// POUs/Local/Objects/Primitive/FB_BACnet_INT
// Integer Value Object
{attribute 'enable_dynamic_creation'}
FUNCTION_BLOCK FB_BACnet_INT EXTENDS FB_BACnet_Object
VAR_INPUT CONSTANT PERSISTENT
	{region 'Operational Parameters'}
		{attribute 'parameterCategory':='Value'}
		nValue : DINT;
		{attribute 'parameterCategory':='Value'}
		eUnit : E_BA_Unit := E_BA_Unit.eOther_NoUnits;
	{endregion}
END_VAR
VAR_OUTPUT
	nPresVal : DINT;
END_VAR

IF bReady THEN
	nPresVal := nValue;
ELSE
	nPresVal := 0;
END_IF

SUPER^();

METHOD PROTECTED OnObjectStateChanged
SUPER^.OnObjectStateChanged();

CASE (tState) OF
	TCOM_STATE.TCOM_STATE_PREOP:
		// SyncHandler:
		RequestSyncHandlers(2, 2);

	TCOM_STATE.TCOM_STATE_SAFEOP:
		SyncProperty(E_BACnetPropIdentifier.PropPresentValue, SIZEOF(nValue), ADR(nValue), 0, eFullSync_InitPLC);
	
	TCOM_STATE.TCOM_STATE_OP:
		SyncProperty(E_BACnetPropIdentifier.PropUnits, SIZEOF(eUnit), ADR(eUnit), 0, eFullSync_InitPLC);
		
END_CASE
END_METHOD

METHOD FB_init : BOOL
VAR_INPUT
	bInitRetains : BOOL; // if TRUE, the retain variables are initialized (warm start / cold start)
	bInCopyCode : BOOL;  // if TRUE, the instance afterwards gets moved into the copy code (online change)
END_VAR
eObjectType := E_BACnetObjType.ObjIntegerValue;
END_METHOD

END_FUNCTION_BLOCK

// POUs/Local/Objects/Primitive/FB_BACnet_LAV
// Large AnalogValue Object
{attribute 'enable_dynamic_creation'}
FUNCTION_BLOCK FB_BACnet_LAV EXTENDS FB_BACnet_Object
VAR_INPUT CONSTANT PERSISTENT
	{region 'Operational Parameters'}
		{attribute 'parameterCategory':='Value'}
		fValue : LREAL;
		{attribute 'parameterCategory':='Value'}
		eUnit : E_BA_Unit := E_BA_Unit.eOther_NoUnits;
	{endregion}
END_VAR
VAR_OUTPUT
	fPresVal : LREAL;
END_VAR

IF bReady THEN
	fPresVal := fValue;
ELSE
	fPresVal := 0;
END_IF

SUPER^();

METHOD PROTECTED OnObjectStateChanged
SUPER^.OnObjectStateChanged();

CASE (tState) OF
	TCOM_STATE.TCOM_STATE_PREOP:
		// SyncHandler:
		RequestSyncHandlers(2, 2);

	TCOM_STATE.TCOM_STATE_SAFEOP:
		SyncProperty(E_BACnetPropIdentifier.PropPresentValue, SIZEOF(fValue), ADR(fValue), 0, eFullSync_InitPLC);
	
	TCOM_STATE.TCOM_STATE_OP:
		SyncProperty(E_BACnetPropIdentifier.PropUnits, SIZEOF(eUnit), ADR(eUnit), 0, eFullSync_InitPLC);
		
END_CASE
END_METHOD

METHOD FB_init : BOOL
VAR_INPUT
	bInitRetains : BOOL; // if TRUE, the retain variables are initialized (warm start / cold start)
	bInCopyCode : BOOL;  // if TRUE, the instance afterwards gets moved into the copy code (online change)
END_VAR
eObjectType := E_BACnetObjType.ObjLargeAnalogValue;
END_METHOD

END_FUNCTION_BLOCK

// POUs/Local/Objects/Primitive/FB_BACnet_String
// Integer Value Object
{attribute 'enable_dynamic_creation'}
FUNCTION_BLOCK FB_BACnet_String EXTENDS FB_BACnet_Object
VAR_INPUT CONSTANT PERSISTENT
	{region 'Operational Parameters'}
		{attribute 'parameterCategory':='Value'}
		{attribute 'TcEncoding':='UTF-8'}
		sValue : T_MaxString;
	{endregion}
END_VAR

SUPER^();

METHOD PROTECTED OnObjectStateChanged
SUPER^.OnObjectStateChanged();

CASE (tState) OF
	TCOM_STATE.TCOM_STATE_PREOP:
		// SyncHandler:
		RequestSyncHandlers(1, 1);

	TCOM_STATE.TCOM_STATE_SAFEOP:
		;
	
	TCOM_STATE.TCOM_STATE_OP:
		SyncProperty(E_BACnetPropIdentifier.PropDescription, SIZEOF(sValue), ADR(sValue), 0, eFullSync_InitPLC);
		
END_CASE
END_METHOD

METHOD FB_init : BOOL
VAR_INPUT
	bInitRetains : BOOL; // if TRUE, the retain variables are initialized (warm start / cold start)
	bInCopyCode : BOOL;  // if TRUE, the instance afterwards gets moved into the copy code (online change)
END_VAR
eObjectType := E_BACnetObjType.ObjCharacterStringValue;
END_METHOD

END_FUNCTION_BLOCK

// POUs/Local/Objects/Primitive/FB_BACnet_UINT
// Large AnalogValue Object
{attribute 'enable_dynamic_creation'}
FUNCTION_BLOCK FB_BACnet_UINT EXTENDS FB_BACnet_Object
VAR_INPUT CONSTANT PERSISTENT
	{region 'Operational Parameters'}
		{attribute 'parameterCategory':='Value'}
		nValue : DINT;
		{attribute 'parameterCategory':='Value'}
		eUnit : E_BA_Unit := E_BA_Unit.eOther_NoUnits;
	{endregion}
END_VAR
VAR_OUTPUT
	nPresVal : LREAL;
END_VAR

IF bReady THEN
	nPresVal := nValue;
ELSE
	nPresVal := 0;
END_IF

SUPER^();

METHOD PROTECTED OnObjectStateChanged
SUPER^.OnObjectStateChanged();

CASE (tState) OF
	TCOM_STATE.TCOM_STATE_PREOP:
		// SyncHandler:
		RequestSyncHandlers(2, 2);

	TCOM_STATE.TCOM_STATE_SAFEOP:
		SyncProperty(E_BACnetPropIdentifier.PropPresentValue, SIZEOF(nValue), ADR(nValue), 0, eFullSync_InitPLC);
	
	TCOM_STATE.TCOM_STATE_OP:
		SyncProperty(E_BACnetPropIdentifier.PropUnits, SIZEOF(eUnit), ADR(eUnit), 0, eFullSync_InitPLC);
		
END_CASE
END_METHOD

METHOD FB_init : BOOL
VAR_INPUT
	bInitRetains : BOOL; // if TRUE, the retain variables are initialized (warm start / cold start)
	bInCopyCode : BOOL;  // if TRUE, the instance afterwards gets moved into the copy code (online change)
END_VAR
eObjectType := E_BACnetObjType.ObjPositiveIntegerValue;
END_METHOD

END_FUNCTION_BLOCK

// POUs/Local/Objects/FB_BACnet_Acc_IO
// Accumulator Object
// - Terminal communication
{attribute 'pin_presentation_order_outputs' := 'nRawValue'}
FUNCTION_BLOCK FB_BACnet_Acc_IO EXTENDS FB_BACnet_BaseAcc
VAR_OUTPUT
	nPulseRate : UDINT;
END_VAR
VAR_INPUT CONSTANT PERSISTENT
	{region 'Variable Parameters'}
		{attribute 'parameterCategory':='Scale'}		  
		stScale : ST_BACnet_Scale;
		{attribute 'parameterCategory':='Scale'}		  	 
		stPrescale :  ST_BACnet_Prescale;
			  
		{attribute 'parameterCategory':='Value'}
		nValueSet : UDINT;
		{attribute 'parameterCategory':='Value'}
		{attribute 'parameterUnit':= 's'}	 
		nLimitMonitoringInterval : UDINT;		
	{endregion}
END_VAR
VAR PERSISTENT
	{region 'Output-Properties'}	
		{attribute 'parameterCategory':='Value'}
		nValueBeforeChange : UDINT;
		{attribute 'parameterCategory':='Value'}
		stValueChangeTime : ST_BA_DateTime;
	{endregion}
END_VAR
VAR
	{region 'Raw I/O'}
		nRawValue			AT %I*	: UINT;				// Bus terminal value
	{endregion}
END_VAR

SUPER^();

METHOD PROTECTED OnObjectStateChanged
CASE (tState) OF
	TCOM_STATE.TCOM_STATE_PREOP:
		// SyncHandler:
		RequestSyncHandlers(7, 5);
		
		WritePropertyUDInt(E_BACnetPropIdentifier.PropLimitMonitoringInverval, nLimitMonitoringInterval);
		
	TCOM_STATE.TCOM_STATE_SAFEOP:
		SyncProperty(E_BACnetPropIdentifier.PropRawIoAccumulatorUnsignedValue, SIZEOF(nRawValue), ADR(nRawValue), 0, eSync_ToSupplement);
		SyncProperty(E_BACnetPropIdentifier.PropPulseRate, SIZEOF(nPulseRate), ADR(nPulseRate), 0, eSync_FromSupplement);
		
	TCOM_STATE.TCOM_STATE_OP:
		SyncProperty(E_BACnetPropIdentifier.PropValueBeforeChange, SIZEOF(nValueBeforeChange), ADR(nValueBeforeChange), 0, eSync_FromSupplementInitPLC);
		SyncProperty(E_BACnetPropIdentifier.PropValueChangeTime, SIZEOF(stValueChangeTime), ADR(stValueChangeTime), 0, eSync_FromSupplementInitPLC);
		
		SyncProperty(E_BACnetPropIdentifier.PropLimitMonitoringInverval, SIZEOF(nLimitMonitoringInterval), ADR(nLimitMonitoringInterval), 0, eFullSync_InitPLC);
		SyncProperty(E_BACnetPropIdentifier.PropScale, SIZEOF(stScale), ADR(stScale), 0, eFullSync_InitPLC);
		SyncProperty(E_BACnetPropIdentifier.PropValueSet, SIZEOF(nValueSet), ADR(nValueSet), 0, eFullSync_InitPLC);		
		SyncProperty(E_BACnetPropIdentifier.PropPrescale, SIZEOF(stPrescale), ADR(stPrescale), 0, eFullSync_InitPLC);
		
END_CASE

SUPER^.OnObjectStateChanged();
END_METHOD

PROPERTY ValueBeforeChange : UDINT
GET
ValueBeforeChange := nValueBeforeChange;
END_GET
END_PROPERTY

PROPERTY ValueChangeTime : ST_BA_DateTime
GET
ValueChangeTime := stValueChangeTime;
END_GET
END_PROPERTY

END_FUNCTION_BLOCK

// POUs/Local/Objects/FB_BACnet_Acc_Raw
// Accumulator Object
// - Raw communication
{attribute 'pin_presentation_order_outputs' := 'fPresVal,bEvent,eRlbty'}
{attribute 'enable_dynamic_creation'}
FUNCTION_BLOCK FB_BACnet_Acc_Raw EXTENDS FB_BACnet_BaseAcc
VAR_INPUT
	{region 'Raw I/O'}
		nRawVal						: UINT;				// Raw value
	{endregion}
END_VAR
VAR_OUTPUT
	nPulseRate						: UDINT;
END_VAR
VAR_INPUT CONSTANT PERSISTENT
	{region 'Variable Parameters'}
		{attribute 'parameterCategory':='Scale'}		  
		stScale : ST_BACnet_Scale;
		{attribute 'parameterCategory':='Scale'}		  	 
		stPrescale :  ST_BACnet_Prescale;	
			  
		{attribute 'parameterCategory':='Value'}
		nValueSet : UDINT;
		{attribute 'parameterCategory':='Value'}
		{attribute 'parameterUnit':= 's'}	 
		nLimitMonitoringInterval : UDINT;		
	{endregion}
END_VAR
VAR PERSISTENT
	{region 'Output-Properties'}	
		nValueBeforeChange			: UDINT;
		stValueChangeTime			: ST_BA_DateTime;
	{endregion}
END_VAR

SUPER^();

METHOD PROTECTED OnObjectStateChanged
CASE (tState) OF
	TCOM_STATE.TCOM_STATE_PREOP:
		// SyncHandler:
		RequestSyncHandlers(8, 5);
		
		WritePropertyUDInt(E_BACnetPropIdentifier.PropLimitMonitoringInverval, nLimitMonitoringInterval);

	TCOM_STATE.TCOM_STATE_SAFEOP:
		SyncProperty(E_BACnetPropIdentifier.PropRawIoAccumulatorUnsignedValue, SIZEOF(nRawVal), ADR(nRawVal), 0, eSync_ToSupplement);
		SyncProperty(E_BACnetPropIdentifier.PropPulseRate, SIZEOF(nPulseRate), ADR(nPulseRate), 0, eSync_FromSupplement);
		
	TCOM_STATE.TCOM_STATE_OP:
		SyncProperty(E_BACnetPropIdentifier.PropValueBeforeChange, SIZEOF(nValueBeforeChange), ADR(nValueBeforeChange), 0, eSync_FromSupplementInitPLC);
		SyncProperty(E_BACnetPropIdentifier.PropValueChangeTime, SIZEOF(stValueChangeTime), ADR(stValueChangeTime), 0, eSync_FromSupplementInitPLC);
	
		SyncProperty(E_BACnetPropIdentifier.PropLimitMonitoringInverval, SIZEOF(nLimitMonitoringInterval), ADR(nLimitMonitoringInterval), 0, eFullSync_InitPLC);
		SyncProperty(E_BACnetPropIdentifier.PropScale, SIZEOF(stScale), ADR(stScale), 0, eFullSync_InitPLC);
		SyncProperty(E_BACnetPropIdentifier.PropValueSet, SIZEOF(nValueSet), ADR(nValueSet), 0, eFullSync_InitPLC);		
		SyncProperty(E_BACnetPropIdentifier.PropPrescale, SIZEOF(stPrescale), ADR(stPrescale), 0, eFullSync_InitPLC);
		
END_CASE

SUPER^.OnObjectStateChanged();
END_METHOD

END_FUNCTION_BLOCK

// POUs/Local/Objects/FB_BACnet_AI
// Analog Input Object
// - process value
{attribute 'pin_presentation_order_outputs' := 'fPresVal,bEvent,eRlbty'}
{attribute 'enable_dynamic_creation'}
FUNCTION_BLOCK FB_BACnet_AI EXTENDS FB_BACnet_BaseAI
VAR_INPUT
	fVal						: REAL;				// Process value
	eRlbtyPgm 					: E_BA_Reliability;
END_VAR

SUPER^();

METHOD PROTECTED OnObjectStateChanged
CASE (tState) OF
	TCOM_STATE.TCOM_STATE_PREOP:
		// SyncHandler:
		RequestSyncHandlers(0, 2);
		
		// Properties:
		EnableProperty(E_BACnetPropIdentifier.PropResolution, FALSE);
		EnableProperty(E_BACnetPropIdentifier.PropScaleOffset, FALSE);
	
	TCOM_STATE.TCOM_STATE_SAFEOP:
		SyncProperty(E_BACnetPropIdentifier.PropPresentValue, SIZEOF(fVal), ADR(fVal), 0, eSync_ToSupplement); 
		SyncProperty(E_BACnetPropIdentifier.PropReliability, SIZEOF(eRlbtyPgm), ADR(eRlbtyPgm), 0, eSync_ToSupplement);
		
	TCOM_STATE.TCOM_STATE_OP:
		;

END_CASE

SUPER^.OnObjectStateChanged();
END_METHOD

END_FUNCTION_BLOCK

// POUs/Local/Objects/FB_BACnet_AI_IO
// Analog Input Object
// - Terminal communication
{attribute 'pin_presentation_order_outputs' := 'fPresVal,bEvent,eRlbty'}
FUNCTION_BLOCK FB_BACnet_AI_IO EXTENDS FB_BACnet_BaseAI
VAR_INPUT CONSTANT PERSISTENT
	{region 'Fixed Parameters'}
		{attribute 'parameterCategory':='Hardware'}
		nIoBusNr : BYTE := 16#FF;
	{endregion}
	{region 'Variable Parameters'}
		{attribute 'parameterCategory':='Hardware'}
		fResolution : REAL := 0.1;
		{attribute 'parameterCategory':='Hardware'}
		fScaleOffset : REAL := 0;
	{endregion}
END_VAR
VAR
	{region 'Raw I/O'}
		nRawState			AT %I*	: USINT;			// Bus terminal state
		nRawValue			AT %I*	: INT;				// Bus terminal value
	{endregion}
END_VAR

SUPER^();

METHOD PROTECTED OnObjectStateChanged
CASE (tState) OF
	TCOM_STATE.TCOM_STATE_PREOP:
		// SyncHandler:
		RequestSyncHandlers(3, 4);

		IF (nIoBusNr <> 16#FF) THEN
			WritePropertyByte(E_BACnetPropIdentifier.PropIoBusNr, nIoBusNr);
		END_IF
		
	TCOM_STATE.TCOM_STATE_SAFEOP:
		SyncProperty(E_BACnetPropIdentifier.PropRawIoStateUSINT, SIZEOF(nRawState), ADR(nRawState), 0, eSync_ToSupplement);
		SyncProperty(E_BACnetPropIdentifier.PropRawIoAnalogValueINT, SIZEOF(nRawValue), ADR(nRawValue), 0, eSync_ToSupplement);
		
	TCOM_STATE.TCOM_STATE_OP:
		SyncProperty(E_BACnetPropIdentifier.PropResolution, SIZEOF(fResolution), ADR(fResolution), 0, eFullSync_InitPLC);
		SyncProperty(E_BACnetPropIdentifier.PropScaleOffset, SIZEOF(fScaleOffset), ADR(fScaleOffset), 0, eFullSync_InitPLC);
		
END_CASE

SUPER^.OnObjectStateChanged();
END_METHOD

END_FUNCTION_BLOCK

// POUs/Local/Objects/FB_BACnet_BI
// Binary Input Object
// - process value
{attribute 'pin_presentation_order_outputs' := 'bPresVal,bEvent,eRlbty'}
{attribute 'enable_dynamic_creation'}
FUNCTION_BLOCK FB_BACnet_BI EXTENDS FB_BACnet_BaseBI
VAR_INPUT
	bVal				: BOOL;				// Process value
	eRlbtyPgm 			: E_BA_Reliability;
END_VAR

SUPER^();

METHOD PROTECTED OnObjectStateChanged
SUPER^.OnObjectStateChanged();

CASE (tState) OF
	TCOM_STATE.TCOM_STATE_PREOP:
		// SyncHandler:
		RequestSyncHandlers(0, 2);

	TCOM_STATE.TCOM_STATE_SAFEOP:
		SyncProperty(E_BACnetPropIdentifier.PropPresentValue, SIZEOF(bVal), ADR(bVal), 0, eSync_ToSupplement);
		SyncProperty(E_BACnetPropIdentifier.PropReliability, SIZEOF(eRlbtyPgm), ADR(eRlbtyPgm), 0, eSync_ToSupplement);
			
	TCOM_STATE.TCOM_STATE_OP:
		;

END_CASE
END_METHOD

END_FUNCTION_BLOCK

// POUs/Local/Objects/FB_BACnet_BI_IO
// Binary Input Object
// - Terminal communication
{attribute 'pin_presentation_order_outputs' := 'bPresVal,bEvent,eRlbty'}
FUNCTION_BLOCK FB_BACnet_BI_IO EXTENDS FB_BACnet_BaseBI
VAR
	{region 'Fixed Parameters'}
		{attribute 'parameterCategory':='Hardware'}
		nIoBusNr : BYTE := 16#FF;
	{endregion}
	{region 'Raw I/O'}
		bRawValue			AT %I*	: BOOL;				// Bus terminal value
	{endregion}
END_VAR

SUPER^();

METHOD PROTECTED OnObjectStateChanged
SUPER^.OnObjectStateChanged();

CASE (tState) OF
	TCOM_STATE.TCOM_STATE_PREOP:
		// SyncHandler:
		RequestSyncHandlers(0, 1);

		IF (nIoBusNr <> 16#FF) THEN
			WritePropertyByte(E_BACnetPropIdentifier.PropIoBusNr, nIoBusNr);
		END_IF
		
	TCOM_STATE.TCOM_STATE_SAFEOP:
		SyncProperty(E_BACnetPropIdentifier.PropRawIoBinaryValueBOOL, SIZEOF(bRawValue), ADR(bRawValue), 0, eSync_ToSupplement);
		
	TCOM_STATE.TCOM_STATE_OP:
		;
		
END_CASE
END_METHOD

END_FUNCTION_BLOCK

// POUs/Local/Objects/FB_BACnet_EE
// Calendar Object
{attribute 'enable_dynamic_creation'}
FUNCTION_BLOCK FB_BACnet_EE EXTENDS FB_BACnet_EventObject 
VAR_INPUT CONSTANT PERSISTENT
	{region 'Variable Parameters'}
		{attribute 'parameterCategory':='Value'}
		stEventParameter : ST_BACnet_EventParameter;
		{attribute 'parameterCategory':='Config'}
		stObjectPropertyReference : ST_BACnet_ObjectPropertyReference;
	{endregion}
END_VAR
VAR_INPUT CONSTANT
	{region 'Variable Parameters'}
		{attribute 'parameterCategory':='Value'}
		bWriteEventParameter : BOOL;
	{endregion}
END_VAR
VAR	
	{region 'COV'}
		bEventParameterChanged	: BOOL;
	{endregion}
END_VAR

IF (bWriteEventParameter) THEN
	WriteContent();
	bWriteEventParameter := FALSE;
END_IF
IF (bEventParameterChanged) THEN
	ReadContent();
	bEventParameterChanged := FALSE;
END_IF

SUPER^();

METHOD PROTECTED OnObjectStateChanged
SUPER^.OnObjectStateChanged();

CASE (tState) OF
	TCOM_STATE.TCOM_STATE_PREOP:
		// SyncHandler:
		RequestSyncHandlers(1, 0);

	TCOM_STATE.TCOM_STATE_SAFEOP:
		;
		
	TCOM_STATE.TCOM_STATE_OP:
		// Validate referred property:
		IF (ValidateReference(stObjectPropertyReference.iObject, stObjectPropertyReference.tObjectID, 16#FF)) THEN
			ObjectPropertyReference := stObjectPropertyReference;
		END_IF
	
		SyncPropertyCOV(E_BACnetPropIdentifier.PropEventParameters, ADR(bEventParameterChanged));
		WriteContent();	
		
END_CASE
END_METHOD

METHOD ReadContent : BOOL
ReadContent := (ReadPropertyEventParameter(stEventParameter) = S_OK);
END_METHOD

METHOD WriteContent : BOOL
WriteContent := (WritePropertyEventParameter(stEventParameter) = S_OK);
END_METHOD

PROPERTY ObjectPropertyReference : ST_BACnet_ObjectPropertyReference
GET
ObjectPropertyReference := stObjectPropertyReference;
END_GET
SET
stObjectPropertyReference := ObjectPropertyReference;

WritePropertyReference(E_BACnetPropIdentifier.PropObjectPropertyReference, stObjectPropertyReference);
END_SET
END_PROPERTY

METHOD FB_init : BOOL
VAR_INPUT
	bInitRetains : BOOL; // if TRUE, the retain variables are initialized (warm start / cold start)
	bInCopyCode : BOOL;  // if TRUE, the instance afterwards gets moved into the copy code (online change)
END_VAR
eObjectType := E_BACnetObjType.ObjEventEnrollment;
END_METHOD

END_FUNCTION_BLOCK

// POUs/Local/Objects/FB_BACnet_ELog
// Event Log Object
FUNCTION_BLOCK FB_BACnet_ELog EXTENDS FB_BACnet_BaseTLog
VAR_INPUT CONSTANT PERSISTENT
	{region 'Fixed Parameters'}
		{attribute 'parameterCategory':='Config'}
		nProcessId : UDINT;
	{endregion}
END_VAR
VAR
	{region 'Buffers'}
		{attribute 'conditionalshow'}
		fbLogBuffer				: FB_BACnet_EventLogBuffer	:= (iRefObject := THIS^);
	{endregion}
END_VAR

// Synchronize Buffers:
fbLogBuffer();

SUPER^();

METHOD PROTECTED OnObjectStateChanged
SUPER^.OnObjectStateChanged();

CASE (tState) OF
	TCOM_STATE.TCOM_STATE_PREOP:
		// SyncHandler:
		RequestSyncHandlers(1, 1);
		
		IF (nProcessId = 0) THEN
			EnableProperty(E_BACnetPropIdentifier.PropProcessId, FALSE);
		END_IF
		
	TCOM_STATE.TCOM_STATE_SAFEOP:
		;

	TCOM_STATE.TCOM_STATE_OP:
		IF (nProcessId <> 0) THEN
			SyncProperty(E_BACnetPropIdentifier.PropProcessId, SIZEOF(nProcessId), ADR(nProcessId), 0, eFullSync_InitPLC);
		END_IF
END_CASE

// Synchronize:
fbLogBuffer.OnObjectStateChanged(tState);
END_METHOD

METHOD FB_init : BOOL
VAR_INPUT
	bInitRetains : BOOL; // if TRUE, the retain variables are initialized (warm start / cold start)
	bInCopyCode : BOOL;  // if TRUE, the instance afterwards gets moved into the copy code (online change)
END_VAR
eObjectType := E_BACnetObjType.ObjEventLog;
END_METHOD

END_FUNCTION_BLOCK

// POUs/Local/Objects/FB_BACnet_Loop_Ref
// Loop Object
{attribute 'enable_dynamic_creation'}
FUNCTION_BLOCK FB_BACnet_Loop_Ref EXTENDS FB_BACnet_BaseLoop
VAR_OUTPUT
	fSetpoint				: REAL;
	fCtrlVar				: REAL;
END_VAR
VAR_INPUT CONSTANT PERSISTENT
	{region 'Variable Parameters'}
		{attribute 'parameterCategory':='Config'}
		stControlledVariableReference : ST_BACnet_ObjectPropertyReference;
		{attribute 'parameterCategory':='Config'}
		stSetpointReference : ST_BACnet_ObjectPropertyReference;
		{attribute 'parameterCategory':='Config'}
		stManipulatedVariableReference : ST_BACnet_ObjectPropertyReference;
	{endregion}
END_VAR

SUPER^();

METHOD PROTECTED OnObjectStateChanged
SUPER^.OnObjectStateChanged();

CASE (tState) OF
	TCOM_STATE.TCOM_STATE_PREOP:
		// SyncHandler:
		RequestSyncHandlers(2, 0);
		
	TCOM_STATE.TCOM_STATE_SAFEOP:
		;
		
	TCOM_STATE.TCOM_STATE_OP:
		// Validate referred properties:
		IF (ValidateReference(stManipulatedVariableReference.iObject, stManipulatedVariableReference.tObjectID, 16#FF)) THEN
			ManipulatedVariableReference := stManipulatedVariableReference;
		END_IF
		IF (ValidateReference(stControlledVariableReference.iObject, stControlledVariableReference.tObjectID, 16#FF)) THEN
			ControlledVariableReference := stControlledVariableReference;
		END_IF
		IF (ValidateReference(stSetpointReference.iObject, stSetpointReference.tObjectID, 16#FF)) THEN
			SetpointReference := stSetpointReference;
		END_IF
		
		SyncProperty(E_BACnetPropIdentifier.PropSetpoint, SIZEOF(fSetpoint), ADR(fSetpoint), 0, eSync_FromSupplement);
		SyncProperty(E_BACnetPropIdentifier.PropControlledVariableValue, SIZEOF(fCtrlVar), ADR(fCtrlVar), 0, eSync_FromSupplement);
	
END_CASE
END_METHOD

PROPERTY ControlledVariable : REAL
GET
ControlledVariable := fCtrlVar;
END_GET
END_PROPERTY

PROPERTY ControlledVariableReference : ST_BACnet_ObjectPropertyReference
GET
ControlledVariableReference := stControlledVariableReference;
END_GET
SET
stControlledVariableReference := ControlledVariableReference;

WritePropertyReference(E_BACnetPropIdentifier.PropControlledVariableReference, stControlledVariableReference);
END_SET
END_PROPERTY

PROPERTY ManipulatedVariableReference : ST_BACnet_ObjectPropertyReference
GET
ManipulatedVariableReference := stManipulatedVariableReference;
END_GET
SET
stManipulatedVariableReference := ManipulatedVariableReference;

WritePropertyReference(E_BACnetPropIdentifier.PropManipulatedVariableReference, stManipulatedVariableReference);
END_SET
END_PROPERTY

PROPERTY Setpoint : REAL
GET
Setpoint := fSetpoint;
END_GET
END_PROPERTY

PROPERTY SetpointReference : ST_BACnet_ObjectPropertyReference
GET
SetpointReference := stSetpointReference;
END_GET
SET
stSetpointReference := SetpointReference;

WritePropertyReference(E_BACnetPropIdentifier.PropSetpointReference, stSetpointReference);
END_SET
END_PROPERTY

END_FUNCTION_BLOCK

// POUs/Local/Objects/FB_BACnet_MI
// Multistate Input Object
// - process value
{attribute 'pin_presentation_order_outputs' := 'nPresVal,bEvent,eRlbty'}
{attribute 'enable_dynamic_creation'}
FUNCTION_BLOCK FB_BACnet_MI EXTENDS FB_BACnet_BaseMI
VAR_INPUT		
	nVal			: UDINT				:= 1;			// Process Value
	eRlbtyPgm 		: E_BA_Reliability;
END_VAR

SUPER^();

METHOD PROTECTED OnObjectStateChanged
SUPER^.OnObjectStateChanged();

CASE (tState) OF
	TCOM_STATE.TCOM_STATE_PREOP:
		// SyncHandler:
		RequestSyncHandlers(0, 2);
		
	TCOM_STATE.TCOM_STATE_SAFEOP:
		SyncProperty(E_BACnetPropIdentifier.PropReliability, SIZEOF(eRlbtyPgm), ADR(eRlbtyPgm), 0, eSync_ToSupplement);
		SyncProperty(E_BACnetPropIdentifier.PropPresentValue, SIZEOF(nVal), ADR(nVal), 0, eSync_ToSupplement);
		
	TCOM_STATE.TCOM_STATE_OP:
		;
		
END_CASE
END_METHOD

END_FUNCTION_BLOCK

// POUs/Local/Objects/FB_BACnet_MI_IO
// Multistate Input Object
// - Terminal communication
{attribute 'pin_presentation_order_outputs' := 'nPresVal,bEvent,eRlbty'}
FUNCTION_BLOCK FB_BACnet_MI_IO EXTENDS FB_BACnet_BaseMI
VAR_INPUT CONSTANT PERSISTENT
	{region 'Variable Parameters'}
		{attribute 'parameterCategory':='Config'}
		eMappingMode : E_BA_ByteMappingMode := E_BA_ByteMappingMode.eIndex1N;
		
		// Used value when no raw-value is active.
		// Note: The mapped process value is shifted '+1' when it is higher than this default value.
		//       > In fact the default value sorts into the range of valid process values.
		{attribute 'parameterCategory':='Value'}
		nRelinquishDefault : UDINT := 1;
	{endregion}
END_VAR
VAR
	{region 'Raw I/O'}
		bRawValue		AT %I*	: ST_BA_Byte;				// Bus terminal value
	{endregion}
	{region 'Internal'}
		{attribute 'conditionalshow'}
		bLastRawValue			: BYTE;
		{attribute 'conditionalshow'}
		nProcVal				: UDINT;
	{endregion}
END_VAR
VAR_STAT
	{region 'Temporary'}
		{attribute 'hide'}
		_bRawValue				: POINTER TO BYTE;
	{endregion}
END_VAR

_bRawValue := ADR(bRawValue);

IF bReady THEN	
	// Trigger change of value:
	IF (_bRawValue^ <> bLastRawValue) THEN
		bLastRawValue := _bRawValue^;
		F_BA_MapUDIFromRawByte(nProcVal, ADR(bRawValue), eMappingMode, nRelinquishDefault);
	END_IF
ELSE
	// Set last value to a different value compared to actual raw value (So a COV is triggered when current instance becomes ready):
	bLastRawValue := (_bRawValue^+1);
	
	nProcVal := nRelinquishDefault;
END_IF

SUPER^();

METHOD PROTECTED OnObjectStateChanged
SUPER^.OnObjectStateChanged();

CASE (tState) OF
	TCOM_STATE.TCOM_STATE_PREOP:
		// SyncHandler:
		RequestSyncHandlers(0, 1);
		
	TCOM_STATE.TCOM_STATE_SAFEOP:
		SyncProperty(E_BACnetPropIdentifier.PropPresentValue, SIZEOF(nProcVal), ADR(nProcVal), 0, eSync_ToSupplement);
		
	TCOM_STATE.TCOM_STATE_OP:
		;
		
END_CASE
END_METHOD

END_FUNCTION_BLOCK

// POUs/Local/Objects/FB_BACnet_PC_Raw
// Pulse Converter Object
{attribute 'enable_dynamic_creation'}
FUNCTION_BLOCK FB_BACnet_PC_Raw EXTENDS FB_BACnet_BasePC
VAR_INPUT
	nRawVal : UINT;
END_VAR

SUPER^();

METHOD PROTECTED OnObjectStateChanged
SUPER^.OnObjectStateChanged();

CASE (tState) OF
	TCOM_STATE.TCOM_STATE_PREOP:
		// SyncHandler:
		RequestSyncHandlers(0, 1);
		
		EnableProperty(E_BACnetPropIdentifier.PropInputReference, FALSE);	
	
		SyncProperty(E_BACnetPropIdentifier.PropRawIoPulseConverterUnsignedValue, SIZEOF(UINT), ADR(nRawVal), 0, eSync_ToSupplement);	
		
	TCOM_STATE.TCOM_STATE_SAFEOP:
		;
		
	TCOM_STATE.TCOM_STATE_OP:
		;

END_CASE
END_METHOD

METHOD FB_init : BOOL
VAR_INPUT
	bInitRetains : BOOL; // if TRUE, the retain variables are initialized (warm start / cold start)
	bInCopyCode : BOOL;  // if TRUE, the instance afterwards gets moved into the copy code (online change)
END_VAR
eObjectType := E_BACnetObjType.ObjPulseConverter;
END_METHOD

END_FUNCTION_BLOCK

// POUs/Local/Objects/FB_BACnet_TLM
FUNCTION_BLOCK FB_BACnet_TLM EXTENDS FB_BACnet_BaseTLog
VAR_INPUT CONSTANT PERSISTENT
	{region 'Variable Parameters'}
		{attribute 'parameterCategory':='Config'}
		aObjectPropertyReferences : ARRAY[1 .. BACnet_Param.nTLM_ReferenceCount] OF ST_BACnet_ObjectPropertyReference;
	{endregion}
END_VAR
VAR
	{region 'Buffers'}
		{attribute 'conditionalshow'}
		fbLogBuffer					: FB_BACnet_TLMBuffer			:= (iRefObject := THIS^);
	{endregion}
END_VAR

// Synchronize Buffers:
fbLogBuffer();

SUPER^();

METHOD PROTECTED OnObjectStateChanged
VAR
	i : DINT;
	_bResult : BOOL;
END_VAR
SUPER^.OnObjectStateChanged();

CASE (tState) OF
	TCOM_STATE.TCOM_STATE_PREOP:
		
		RequestSyncHandlers(1, 1);
	
	TCOM_STATE.TCOM_STATE_SAFEOP:
		;
		
	TCOM_STATE.TCOM_STATE_OP:
		// Validate referred properties:
		FOR i:= 1 TO TO_DINT(BACnet_Param.nTLM_ReferenceCount) DO
			ValidateReference(aObjectPropertyReferences[i].iObject, aObjectPropertyReferences[i].tObjectID, 16#FF);
		END_FOR
		ObjectPropertyReferences := aObjectPropertyReferences;
		
END_CASE

// Synchronize:
fbLogBuffer.OnObjectStateChanged(tState);
END_METHOD

PROPERTY ObjectPropertyReferences : ARRAY[1 .. BACnet_Param.nTLM_ReferenceCount] OF ST_BACnet_ObjectPropertyReference
GET
ObjectPropertyReferences := aObjectPropertyReferences;
END_GET
SET
aObjectPropertyReferences := ObjectPropertyReferences;

{warning disable C0196}
WritePropertyReferenceList(E_BACnetPropIdentifier.PropLogDeviceObjectProperty, aObjectPropertyReferences);
{warning restore C0196}
END_SET
END_PROPERTY

METHOD FB_init : BOOL
VAR_INPUT
	bInitRetains : BOOL; // if TRUE, the retain variables are initialized (warm start / cold start)
	bInCopyCode : BOOL;  // if TRUE, the instance afterwards gets moved into the copy code (online change)
END_VAR
eObjectType := E_BACnetObjType.ObjTrendLogMultiple;
END_METHOD

END_FUNCTION_BLOCK

// POUs/Local/Objects/FB_BACnet_TLog
FUNCTION_BLOCK FB_BACnet_TLog EXTENDS FB_BACnet_BaseTLog
VAR_INPUT CONSTANT PERSISTENT
	{region 'Variable Parameters'}
		{attribute 'parameterCategory':='Config'}
		stObjectPropertyReference : ST_BACnet_ObjectPropertyReference;
		{attribute 'parameterCategory':='Config'}
		bAlignIntervals : BOOL;
		{attribute 'parameterCategory':='Config'}	
		nIntervalOffset : UDINT;
		{attribute 'parameterCategory':='Config'}	
		stClientCOV : ST_BACnet_ClientCOV;
		{attribute 'parameterCategory':='Config'}	
		{attribute 'parameterUnit':= 's'}
		nCOVResubscriptionInterval : UDINT := 3600;
	{endregion}
END_VAR
VAR
	{region 'Buffers'}
		{attribute 'conditionalshow'}
		fbLogBuffer					: FB_BACnet_TrendLogBuffer			:= (iRefObject := THIS^);
	{endregion}
END_VAR

// Synchronize Buffers:
fbLogBuffer();

SUPER^();

METHOD PROTECTED OnObjectStateChanged
SUPER^.OnObjectStateChanged();

CASE (tState) OF
	TCOM_STATE.TCOM_STATE_PREOP:
		// SyncHandler:
		RequestSyncHandlers(5, 5);
		
	TCOM_STATE.TCOM_STATE_SAFEOP:
		;
		
	TCOM_STATE.TCOM_STATE_OP:
		SyncProperty(E_BACnetPropIdentifier.PropAlignIntervals, SIZEOF(bAlignIntervals), ADR(bAlignIntervals), 0, eFullSync_InitPLC);
		SyncProperty(E_BACnetPropIdentifier.PropIntervalOffset, SIZEOF(nIntervalOffset), ADR(nIntervalOffset), 0, eFullSync_InitPLC);
		SyncProperty(E_BACnetPropIdentifier.PropClientCovIncrement, SIZEOF(ST_BACnet_ClientCOV), ADR(stClientCOV), 0, eFullSync_InitPLC);
		SyncProperty(E_BACnetPropIdentifier.PropCovResubscriptionInterval, SIZEOF(nCOVResubscriptionInterval), ADR(nCOVResubscriptionInterval), 0, eFullSync_InitPLC);
		// Validate referred property:
		IF (ValidateReference(stObjectPropertyReference.iObject, stObjectPropertyReference.tObjectID, 16#FF)) THEN
			ObjectPropertyReference := stObjectPropertyReference;
		END_IF
		
END_CASE

fbLogBuffer.OnObjectStateChanged(tState);
END_METHOD

PROPERTY ObjectPropertyReference : ST_BACnet_ObjectPropertyReference
GET
ObjectPropertyReference := stObjectPropertyReference;
END_GET
SET
stObjectPropertyReference := ObjectPropertyReference;

WritePropertyReference(E_BACnetPropIdentifier.PropLogDeviceObjectProperty, stObjectPropertyReference);
END_SET
END_PROPERTY

METHOD FB_init : BOOL
VAR_INPUT
	bInitRetains : BOOL; // if TRUE, the retain variables are initialized (warm start / cold start)
	bInCopyCode : BOOL;  // if TRUE, the instance afterwards gets moved into the copy code (online change)
END_VAR
eObjectType := E_BACnetObjType.ObjTrendLog;
END_METHOD

END_FUNCTION_BLOCK

// POUs/Remote/Objects/Basic/[Base]/Basic/FB_BACnetRM_Object
FUNCTION_BLOCK FB_BACnetRM_Object EXTENDS FB_BACnetRM_BaseObject IMPLEMENTS I_BACnetRM_Object, I_BACnetRM_ObjectOwner
VAR
	{region 'Internal'}
		{attribute 'hide'}
		bParentInit					: BOOL := TRUE;
		{attribute 'hide'}
		fbLogMsg					: FB_BA_LogMessage;
	{endregion}
END_VAR

SUPER^();

// Unused - Implemented for compatibility reason!
{attribute 'hide'}
METHOD OnBACnetRMObjectCOV
VAR_INPUT
	ePropID		: E_BACnetPropIdentifier;
END_VAR
END_METHOD

// Unused - Implemented for compatibility reason!
{attribute 'hide'}
METHOD OnBACnetRMObjectStateChanged
END_METHOD

{attribute 'suppress_wrn_C0410'}
{attribute 'hide'}
PROPERTY LogMsg : REFERENCE TO FB_BA_LogMessage
GET
LogMsg REF= fbLogMsg;
END_GET
END_PROPERTY

METHOD FB_init : BOOL
VAR_INPUT
	bInitRetains : BOOL; // if TRUE, the retain variables are initialized (warm start / cold start)
	bInCopyCode : BOOL;  // if TRUE, the instance afterwards gets moved into the copy code (online change)
END_VAR
iOwner := THIS^;
END_METHOD

END_FUNCTION_BLOCK

// POUs/Remote/Objects/Basic/[Internal]/FB_BACnetRM_BaseObject
{attribute 'no_assign'}
FUNCTION_BLOCK FB_BACnetRM_BaseObject IMPLEMENTS I_BACnetRM_BaseObject
VAR_INPUT CONSTANT
	{region 'Fixed Parameters'}
		{attribute 'parameterCategory':='General'}
		{attribute 'no_copy'}
		Client : REFERENCE TO FB_BACnet_Client;
		{attribute 'parameterCategory':='General'}
		nObjectInstance : UDINT := BACnet_Globals.nBACnetInstId_Auto;	
		{attribute 'parameterCategory':='Communication'}
		eReadMode : E_BACnet_CommMode := E_BACnet_CommMode.eAuto;
	{endregion}
END_VAR
VAR_OUTPUT
	bReady					: BOOL;
END_VAR
VAR
	{region 'SubInit'}
		eObjectType			: E_BACnetObjType				:= 16#FFFF;
		{attribute 'hide'}
		iOwner				: I_BACnetRM_ObjectOwner;												// Owner of current Instance (Pointer to current instance per default)
	{endregion}
END_VAR
VAR
	{region 'General'}
		eErrorID			: E_BACnet_Error				:= E_BACnet_Error.eNoError;
			 
		tObjectID			: T_BACnet_ObjectIdentifier		:= 16#FFFFFFFF;
			 
		{attribute 'hide'}
		{attribute 'no_copy'}
		bInit				: BOOL;
	{endregion}
END_VAR

IF (NOT bReady) THEN
	IF (iOwner = 0) THEN
		eErrorID := E_BACnet_Error.eInvalidParameter;
		F_BA_LogMessage(ADSLOG_MSGTYPE_ERROR, 'O04', 'Owner of BACnet remote-object not defined!');
		
	ELSIF (__ISVALIDREF(Client)) THEN
		IF (NOT Client.bConnected) THEN		
			; // Wait for referred client to be conntected.
		ELSE
			IF NOT bInit THEN
				bInit := TRUE;
				OnObjectStateChanged();
				tObjectID := F_BACnet_GetObjId(eObjectType, nObjectInstance);		
				Client.UpdateRequests();
			ELSE
				IF Client.bReady THEN
					eErrorID := E_BACnet_Error.eNoError;
					bReady := TRUE;
				END_IF
			END_IF
		END_IF
	ELSE
		eErrorID := E_BACnet_Error.eInvalidClient;
		iOwner.LogMsg.Show(ADSLOG_MSGTYPE_ERROR, 'O17', 'Assigned client-reference is invalid!', FALSE);
	END_IF
ELSE
	IF NOT Client.bReady THEN
		bReady := FALSE;
	END_IF
END_IF

{attribute 'hide'}
METHOD OnCOV
VAR_INPUT
	ePropID		: E_BACnetPropIdentifier;
END_VAR
// Notify owner:
iOwner.OnBACnetRMObjectCOV(ePropID);
END_METHOD

{attribute 'hide'}
METHOD OnReqError
VAR_INPUT
	iRequest		: I_BACnetRM_BaseReq;
	stResult		: POINTER TO SendDataRequestResult;
	sLogCode		: STRING			:= '';
END_VAR
VAR_STAT
	{attribute 'hide'}
	_sTemp			: STRING;
	{attribute 'hide'}
	fbMessage		: FB_BA_DecorMessage;
END_VAR
fbMessage.Reset();

IF (stResult = 0) THEN
	iOwner.LogMsg.Show(ADSLOG_MSGTYPE_ERROR, 'ORE04', 'Internal error in implementation of error-handling!', FALSE);
ELSE
	CASE (stResult^.errorType) OF
		E_BACnet_ErrorType.eError:
			IF (NOT F_BACnet_IsErrorClassValid(TO_INT(stResult^.errorClass))) THEN
				iOwner.LogMsg.Show1(ADSLOG_MSGTYPE_ERROR, 'ORE07', 'Received unknown error of invalid class "%d"!', F_DINT(stResult^.errorClass), FALSE);
			ELSIF (NOT F_BACnet_IsErrorCodeValid(TO_INT(stResult^.errorCode))) THEN
				iOwner.LogMsg.Show1(ADSLOG_MSGTYPE_ERROR, 'ORE09', 'Received unknown error of invalid code "%d"!', F_DINT(stResult^.errorCode), FALSE);
			ELSE
				fbMessage.FormatText1('Received error "%s"', F_STRINGEx(BACnet_Globals.aSpec_ErrorCode[stResult^.errorCode]));
				fbMessage.AddDecor1('Class: %s', F_STRINGEx(BACnet_Globals.aSpec_ErrorClass[stResult^.errorClass]));
			END_IF
			
		E_BACnet_ErrorType.eReject:
			IF (NOT F_BACnet_IsRejectReasonValid(TO_INT(stResult^.rejectCode))) THEN
				iOwner.LogMsg.Show1(ADSLOG_MSGTYPE_ERROR, 'ORE16', 'Received unknown rejection of invalid reason "%d"!', F_DINT(stResult^.rejectCode), FALSE);
			ELSE
				fbMessage.FormatText1('Received rejection "%s".', F_STRINGEx(BACnet_Globals.aSpec_RejectReason[stResult^.rejectCode]));
			END_IF
		
		E_BACnet_ErrorType.eAbort:
			IF (NOT F_BACnet_IsAbortReasonValid(TO_INT(stResult^.abortReason))) THEN
				iOwner.LogMsg.Show1(ADSLOG_MSGTYPE_ERROR, 'ORE23', 'Received unknown abort of invalid reason "%d"!', F_DINT(stResult^.abortReason), FALSE);
			ELSE
				fbMessage.FormatText1('Received abort "%s".', F_STRINGEx(BACnet_Globals.aSpec_AbortReason[stResult^.abortReason]));
			END_IF
		
	ELSE
		iOwner.LogMsg.Show1(ADSLOG_MSGTYPE_ERROR, 'ORE29', 'Invalid error of type "%d" received!', F_DINT(stResult^.errorType), FALSE);
	END_CASE
END_IF

IF (NOT fbMessage.IsEmpty) THEN
	// Add further information:
	IF (bReady) THEN
		_sTemp := F_BACnet_GetObjectIdString(tObjectID);
		fbMessage.AddDecor2('Remote Object: [%d]%s', F_UDINT(Client.nDeviceInstance), F_STRINGEx(_sTemp));
	END_IF
	CASE (stResult^.errorClass) OF
		E_BACnet_ErrorClass.eProperty:
			fbMessage.AddDecor1('Property: %d', F_INT(stResult^.propertyIdentifier));
//		E_BACnet_ErrorClass.xxx:
//			fbMessage.AddDecor1('Invoke ID: %d', F_UDINT(stResult^.invokeId));
//		E_BACnet_ErrorClass.xxx:
//			fbMessage.AddDecor1('Process ID: %d', F_UDINT(stResult^.processId));
	END_CASE
	
	// Build message:
	IF (fbMessage.Finish()) THEN
		iOwner.LogMsg.Show(ADSLOG_MSGTYPE_ERROR, sLogCode, fbMessage.sOutput, TRUE);
	END_IF
END_IF
END_METHOD

METHOD PROTECTED OnObjectStateChanged
// Notify owner:
iOwner.OnBACnetRMObjectStateChanged();
END_METHOD

PROPERTY Error : BOOL
GET
Error := (eErrorID <> E_BACnet_Error.eNoError);
END_GET
END_PROPERTY

PROPERTY ObjectID : T_BACnet_ObjectIdentifier
GET
ObjectID := tObjectID;
END_GET
END_PROPERTY

PROPERTY ObjectInstance : UDINT
GET
ObjectInstance := nObjectInstance;
END_GET
SET
PUBLIC 
VAR
END_VAR
nObjectInstance:=ObjectInstance;
tObjectID := F_BACnet_GetObjId(eObjectType, nObjectInstance);
END_SET
END_PROPERTY

PROPERTY ObjectType : E_BACnetObjType
GET
ObjectType := eObjectType;
END_GET
SET
PUBLIC 
VAR
END_VAR
eObjectType:=ObjectType;
tObjectID := F_BACnet_GetObjId(eObjectType, nObjectInstance);
END_SET
END_PROPERTY

PROPERTY ReadMode : E_BACnet_CommMode
GET
ReadMode:=eReadMode;
END_GET
SET
eReadMode:=ReadMode;
END_SET
END_PROPERTY

METHOD SyncProperty : BOOL
VAR_INPUT
	ePropID		: E_BACnetPropIdentifier;
	nSize		: UDINT;
	pData		: PVOID;
	eSyncMode	: E_BA_SyncModeRM;
END_VAR
VAR_STAT
	{attribute 'hide'}
	stRdEntry	: POINTER TO ST_BACnetRM_ReadEntry;
	{attribute 'hide'}
	stWrtEntry	: POINTER TO ST_BACnetRM_WriteEntry;
END_VAR
SyncProperty:=SyncPropertyReal(ePropID, nSize, pData, eSyncMode, 0.0);
END_METHOD

METHOD SyncPropertyEnable : BOOL
VAR_INPUT
	ePropID		: E_BACnetPropIdentifier;
	nSize		: UDINT;
	pData		: PVOID;
	pEnable		: POINTER TO BOOL := 0;
	eSyncMode	: E_BA_SyncModeRM;
END_VAR
VAR_STAT
	{attribute 'hide'}
	stWrtEntry	: POINTER TO ST_BACnetRM_WriteEntry;
END_VAR
SyncPropertyEnable:=SyncPropertyPrioReal(ePropID, nSize, pData, pEnable, 0, E_BACnet_Priority.Last, eSyncMode, 0.0);
END_METHOD

METHOD SyncPropertyIdx : BOOL
VAR_INPUT
	ePropID		: E_BACnetPropIdentifier;
	nSize		: UDINT;
	pData		: PVOID;
	nIndex		: INT(0..2);
	eSyncMode	: E_BA_SyncModeRM;
END_VAR
VAR_STAT
	{attribute 'hide'}
	stRdEntry	: POINTER TO ST_BACnetRM_ReadEntry;
	{attribute 'hide'}
	stWrtEntry	: POINTER TO ST_BACnetRM_WriteEntry;
END_VAR
IF (0 <= nIndex) AND_THEN (nIndex <= 2) THEN
	CASE (eSyncMode) OF
		E_BA_SyncModeRM.eRead:
			IF (SyncPropertyIdx := Client.AddReadEntry(THIS^, ePropID, E_BACnet_Priority.Invalid, stResult=>stRdEntry)) THEN
				stRdEntry^.nData := nSize;
				stRdEntry^.pData := pData;
				stRdEntry^.nIndex := TO_UDINT(nIndex);
			END_IF
		
		E_BA_SyncModeRM.eWrite:
			iOwner.LogMsg.Show1(ADSLOG_MSGTYPE_ERROR, 'SPI11', 'Unimplemented Sync-Mode "%d"!', F_INT(eSyncMode), TRUE);
		
	ELSE
		iOwner.LogMsg.Show1(ADSLOG_MSGTYPE_ERROR, 'SPI14', 'Invalid Sync-Mode "%d"!', F_INT(eSyncMode), TRUE);
	END_CASE
ELSE
	iOwner.LogMsg.Show1(ADSLOG_MSGTYPE_ERROR, 'SPI17', 'Invalid parameter "Index=%d"!', F_INT(nIndex), TRUE);
END_IF
END_METHOD

METHOD SyncPropertyPrio : BOOL
VAR_INPUT
	ePropID		: E_BACnetPropIdentifier;
	nSize		: UDINT;
	pData		: PVOID;
	pEnable		: POINTER TO BOOL := 0;
	pNull		: POINTER TO BOOL := 0;
	ePriority	: E_BACnet_Priority := E_BACnet_Priority.Last;
	eSyncMode	: E_BA_SyncModeRM;
END_VAR
VAR_STAT
	{attribute 'hide'}
	stWrtEntry	: POINTER TO ST_BACnetRM_WriteEntry;
END_VAR
SyncPropertyPrio:=SyncPropertyPrioReal(ePropID, nSize, pData, pEnable, pNull, ePriority, eSyncMode, 0.0);
END_METHOD

METHOD SyncPropertyPrioReal : BOOL
VAR_INPUT
	ePropID			: E_BACnetPropIdentifier;
	nSize			: UDINT;
	pData			: PVOID;
	pEnable			: POINTER TO BOOL := 0;
	pNull			: POINTER TO BOOL := 0;
	ePriority		: E_BACnet_Priority := E_BACnet_Priority.Last;
	eSyncMode		: E_BA_SyncModeRM;
	fCOVIncrement	: REAL;
END_VAR
VAR_STAT
	{attribute 'hide'}
	stWrtEntry	: POINTER TO ST_BACnetRM_WriteEntry;
END_VAR
CASE (eSyncMode) OF
	E_BA_SyncModeRM.eRead:
		iOwner.LogMsg.Show1(ADSLOG_MSGTYPE_ERROR, 'SPP03', 'Unimplemented Sync-Mode "%d"!', F_INT(eSyncMode), TRUE);
	
	E_BA_SyncModeRM.eWrite:
		IF (SyncPropertyPrioReal := Client.AddWriteEntry(THIS^, ePropID, ePriority, stResult=>stWrtEntry)) THEN
			stWrtEntry^.nData := nSize;
			stWrtEntry^.pData := pData;
			stWrtEntry^.pEnable := pEnable;
			stWrtEntry^.pNull := pNull;
			stWrtEntry^.nPriority := TO_UDINT(ePriority);
			stWrtEntry^.fCOVIncrement := fCOVIncrement;
		END_IF
	
ELSE
	iOwner.LogMsg.Show1(ADSLOG_MSGTYPE_ERROR, 'SPP09', 'Invalid Sync-Mode "%d"!', F_INT(eSyncMode), TRUE);
END_CASE
END_METHOD

METHOD SyncPropertyReal : BOOL
VAR_INPUT
	ePropID			: E_BACnetPropIdentifier;
	nSize			: UDINT;
	pData			: PVOID;
	eSyncMode		: E_BA_SyncModeRM;
	fCOVIncrement	: REAL;
END_VAR
VAR_STAT
	{attribute 'hide'}
	stRdEntry	: POINTER TO ST_BACnetRM_ReadEntry;
	{attribute 'hide'}
	stWrtEntry	: POINTER TO ST_BACnetRM_WriteEntry;
END_VAR
CASE (eSyncMode) OF
	E_BA_SyncModeRM.eRead:
		IF (SyncPropertyReal := Client.AddReadEntry(THIS^, ePropID, E_BACnet_Priority.Invalid, stResult=>stRdEntry)) THEN
			stRdEntry^.nData := nSize;
			stRdEntry^.pData := pData;
			stRdEntry^.fCOVIncrement := fCOVIncrement;
		END_IF
	
	E_BA_SyncModeRM.eWrite:
		IF (SyncPropertyReal := Client.AddWriteEntry(THIS^, ePropID, E_BACnet_Priority.Invalid, stResult=>stWrtEntry)) THEN
			stWrtEntry^.nData := nSize;
			stWrtEntry^.pData := pData;
			stWrtEntry^.fCOVIncrement := fCOVIncrement;
		END_IF
	
ELSE
	iOwner.LogMsg.Show1(ADSLOG_MSGTYPE_ERROR, 'SP09', 'Invalid Sync-Mode "%d"!', F_INT(eSyncMode), TRUE);
END_CASE
END_METHOD

END_FUNCTION_BLOCK

// TEST/TestPackage/CLIENT
PROGRAM CLIENT
VAR
	fbClient			: FB_BACnet_Client					:= (nDeviceInstance := 3776986(*, eReadMode := E_BACnet_CommMode.eCov*));
	
	AV01				: FB_BACnetRM_AV					:= (Client := fbClient, nObjectInstance:=13011);
	AVDsp				: FB_BACnetRM_AV_Disp				:= (Client := fbClient, nObjectInstance:=10001);
	AVSp				: FB_BACnetRM_AV_Setp				:= (Client := fbClient, nObjectInstance:=10002);
	AI01				: FB_BACnetRM_AI					:= (Client := fbClient, nObjectInstance:=10000);
	AO01				: FB_BACnetRM_AO					:= (Client := fbClient, nObjectInstance:=10000);
	
	BV01				: FB_BACnetRM_BV					:= (Client := fbClient, nObjectInstance:=99);
	BVDsp				: FB_BACnetRM_BV_Disp				:= (Client := fbClient, nObjectInstance:=10001);
	BVSp				: FB_BACnetRM_BV_Setp				:= (Client := fbClient, nObjectInstance:=10002);
	BI01				: FB_BACnetRM_BI					:= (Client := fbClient, nObjectInstance:=10000);
	BO01				: FB_BACnetRM_BO					:= (Client := fbClient, nObjectInstance:=10000);
	
	MV01				: FB_BACnetRM_MV					:= (Client := fbClient, nObjectInstance:=99);
	MVDsp				: FB_BACnetRM_MV_Disp				:= (Client := fbClient, nObjectInstance:=10001);
	MVSp				: FB_BACnetRM_MV_Setp				:= (Client := fbClient, nObjectInstance:=10002);
	MI01				: FB_BACnetRM_MI					:= (Client := fbClient, nObjectInstance:=10000);
	MO01				: FB_BACnetRM_MO					:= (Client := fbClient, nObjectInstance:=10000);
	
	TLog				: FB_BACnetRM_TLog					:= (Client := fbClient, nObjectInstance:=10000);
	TLM					: FB_BACnetRM_TLM					:= (Client := fbClient, nObjectInstance:=10000);
	Cal01				: FB_BACnetRM_Cal					:= (Client := fbClient, nObjectInstance:=10000);
	SchedA				: FB_BACnetRM_SchedA				:= (Client := fbClient, nObjectInstance:=10000);
	SchedB				: FB_BACnetRM_SchedB				:= (Client := fbClient, nObjectInstance:=10001);
	SchedM				: FB_BACnetRM_SchedM				:= (Client := fbClient, nObjectInstance:=10002);
	Loop1				: FB_BACnetRM_Loop					:= (Client := fbClient, nObjectInstance:=10000);
	Loop2				: FB_BACnetRM_CnvLoop				:= (Client := fbClient, nObjectInstance:=10000); 
	File				: FB_BACnetRM_File					:= (Client := fbClient, nObjectInstance:=0);
	
	NC_AlmStd			: FB_BACnetRM_NC					:= (Client := fbClient, nObjectInstance:=11);
	
	Acc					: FB_BACnetRM_Acc					:= (Client := fbClient, nObjectInstance:=10000);
	PC					: FB_BACnetRM_PC					:= (Client := fbClient, nObjectInstance:=10000);
	Prog				: FB_BACnetRM_Prog					:= (Client := fbClient, nObjectInstance:=10000);
END_VAR
VAR
	diag : ST_BACnet_Diagnosis;
	scanRes : ARRAY [0..99] OF ST_BACnetRM_ScanResult;
	syncTime : ST_BA_DateTime;
	
	bDiag : BOOL;
	bScan : BOOL;
	bGet : BOOL;
	bSync : BOOL;
END_VAR

fbClient();

AV01();
AVDsp();
AVSp();
AI01();
AO01();

BV01();
BVDsp();
BVSp();
BI01();
BO01();

MV01();
MVDsp();
MVSp();
MI01();
MO01();

TLog();
TLM();
Cal01();
SchedA();
SchedB();
SchedM();
Loop1();
Loop2();

NC_AlmStd();

Acc();
PC();
Prog();

IF bDiag THEN
	fbClient.Adapter.GetDiagnosis(ADR(diag));
END_IF

IF bScan THEN	
	fbClient.Adapter.StartScan();
	bScan:=FALSE;
END_IF

IF bGet THEN
	fbClient.Adapter.GetScanResult(ADR(scanRes), 100);
	bGet:=FALSE;
END_IF

IF bSync THEN
	fbClient.Adapter.TimeSync(ADR(syncTime), TRUE);
	bSync:=FALSE;
END_IF

END_PROGRAM

// POUs/Remote/FB_BACnet_Client
{attribute 'enable_dynamic_creation'}
{attribute 'no_assign'}
FUNCTION_BLOCK FB_BACnet_Client IMPLEMENTS I_BACnetRM_Object
VAR_INPUT CONSTANT
	{region 'Fixed Parameters'}
		{attribute 'parameterCategory':='General'}
		{attribute 'no_copy'}
		Adapter	: REFERENCE TO FB_BACnet_Adapter := BACnet_Globals.DefaultAdapter;
		{attribute 'parameterCategory':='General'}
		nDeviceInstance : UDINT;
	{endregion}
END_VAR
VAR_INPUT CONSTANT PERSISTENT
	{region 'Variable Parameters'}
		{attribute 'parameterCategory':='Communication'}
		nMaxParallelRequests : UDINT := 1;
		{attribute 'parameterCategory':='Communication'}
		nRPMPropertiesPerRequest : UDINT := 80;
		{attribute 'parameterCategory':='Communication'}
		tCOVLifeTime : TIME := T#240S;	
		{attribute 'parameterCategory':='Communication'}
		eReadMode : E_BACnet_CommMode := E_BACnet_CommMode.eAuto;
		{attribute 'parameterCategory':='Communication'}
		tReadCycleTime : TIME := T#5S;
		{attribute 'parameterCategory':='Communication'}
		tWriteCycleTime : TIME := T#5S;
		{attribute 'parameterCategory':='Supported Services'}
		bSuppRpm  : BOOL;
		{attribute 'parameterCategory':='Supported Services'}
		bSuppCov  : BOOL;
		{attribute 'parameterCategory':='Supported Services'}
		bSuppCovP : BOOL;
	{endregion}
END_VAR
VAR_OUTPUT
	bReady					: BOOL;
	eErrorID				: E_BACnet_Error;
	nAdsPort 				: UINT;
	bConnected  			: BOOL;
END_VAR
VAR
	{region 'General'}
		tObjectID			: T_BACnet_ObjectIdentifier		:= 16#FFFFFFFF;
	{endregion}
END_VAR
VAR
	{region 'General'}
		eState				: E_BACnetRM_ClientState;	
		stSupportedServices	: ST_BACnet_ServicesSupportedBits;
		nMaxApduSize 		: UDINT;
	{endregion}
	{region 'Request Lists'}
		{region 'Read'}
			{attribute 'hide'}
			stReadList 		: POINTER TO ST_BACnetRM_ReadEntry;
			{attribute 'hide'}
			nReadList		: UDINT := 0;
			{attribute 'hide'}
			nReadMax		: UDINT := 0;
		{endregion}
		{region 'Write'}
			{attribute 'hide'}
			stWriteList		: POINTER TO ST_BACnetRM_WriteEntry;
			{attribute 'hide'}
			nWriteList		: UDINT := 0;
			{attribute 'hide'}
			nWriteMax		: UDINT := 0;	
		{endregion}
	{endregion}
	{region 'Request Fifo'}
		{region 'Cyclic'}
			{attribute 'hide'}
			stReqList		: POINTER TO ST_BACnetRM_ReqPtr := 0;
			{attribute 'hide'}
			nReqList		: UDINT := 0;
			{attribute 'hide'}
			nCurReq			: UDINT := 0;
		{endregion}
		{region 'Acyclic / Dynamic'}
			{attribute 'hide'}
			fbReadFifo		: FB_BACnetRM_ReqFifo := (Client := THIS^);
			{attribute 'hide'}
			fbWriteFifo		: FB_BACnetRM_ReqFifo := (Client := THIS^);
		{endregion}
				  
		nOpenReq			: UDINT := 0;
		{attribute 'hide'}
		bUpdateReqs			: BOOL;
	{endregion}
		 
	{region 'Internal'}
		{attribute 'hide'}
		iServer				: ITcIoBACnetPlcServer;
		{attribute 'hide'}
		iClient				: ITcIoBACnetPlcClient;
		{attribute 'hide'}
		iDevice				: ITcIoBACnetPlcDevice;
		{attribute 'hide'}
		_bCreated			: BOOL;
			 
		{attribute 'hide'}
		fbRead				: FB_BACnetRM_ReadProperty := (Client:=THIS^);
		{attribute 'hide'}
		_ClientStatus		: WORD;
		{attribute 'hide'}
		_ClientControl		: WORD;
		{attribute 'hide'}
		_tReInitTime		: TIME;
		{attribute 'hide'}
		_tCycleStartTime	: TIME;
		diagCycleDuration 	: TIME;
	{endregion}
END_VAR
VAR_STAT
	{region 'Temporary'}
		{attribute 'hide'}
		_n					: UDINT;
		{attribute 'hide'}
		_nRpmTreshold		: UDINT;
	{endregion}
END_VAR

IF (__ISVALIDREF(Adapter)) THEN
	Adapter();
	
	IF (iDevice = 0) THEN
		iDevice := Adapter.Device;
	END_IF
END_IF

IF iClient = 0 THEN
	IF iDevice <> 0 THEN
		IF S_OK <> iDevice.GetClientById(nDeviceInstance, ADR(iServer)) THEN
			IF NOT _bCreated THEN
				IF S_OK = iDevice.CreateClient(nDeviceInstance) THEN
					_bCreated := TRUE;
				END_IF
			END_IF			
		ELSE
			iServer.GetAdsPort(ADR(nAdsPort));
			IF S_OK <> iServer.TcQueryInterface(TC_GLOBAL_IID_LIST.IID_ITcIoBACnetPlcClient, ADR(iClient)) THEN
				eErrorID := E_BACnet_Error.eInvalidClient;
			END_IF
		END_IF
	END_IF
END_IF

IF iClient <> 0 THEN
	iServer.UpdateDeviceStatus(ADR(_ClientControl), ADR(_ClientStatus));	
	IF Adapter.bEthLink THEN
		bConnected := NOT (SHR((_ClientStatus AND 16#FF00), 8) < 4);
	ELSE
		bConnected := FALSE;
	END_IF
	CASE eState OF
		E_BACnetRM_ClientState.eInit:
			IF bConnected THEN
				tObjectID := F_BACnet_GetObjId(ObjectType, nDeviceInstance);
				IF stSupportedServices.bSuppReadProperty THEN
					State:=E_BACnetRM_ClientState.eCalcAuto;
				ELSE
					State:=E_BACnetRM_ClientState.eReadSupportedServices;
				END_IF
			END_IF
		E_BACnetRM_ClientState.eReadSupportedServices:
			IF fbRead.bReady OR fbRead.bError THEN
				IF fbRead.bError THEN
					State:=E_BACnetRM_ClientState.eError;
				ELSE
					State:=E_BACnetRM_ClientState.eReadApduSize;
				END_IF
				fbRead(bExecute:=FALSE);
			ELSIF NOT fbRead.bBusy THEN
				fbRead(iObject:=THIS^, ePropID:=E_BACnetPropIdentifier.PropProtocolServicesSupported, nData:=SIZEOF(stSupportedServices), pData:=ADR(stSupportedServices), bExecute:=TRUE);
			END_IF
			fbReadFifo.ProcessReadFifo();
		E_BACnetRM_ClientState.eReadApduSize:
			IF fbRead.bReady OR fbRead.bError THEN
				IF fbRead.bError THEN
					State:=E_BACnetRM_ClientState.eError;
				ELSE
					State:=E_BACnetRM_ClientState.eCalcAuto;
				END_IF
				fbRead(bExecute:=FALSE);
			ELSIF NOT fbRead.bBusy THEN
				fbRead(iObject:=THIS^, ePropID:=E_BACnetPropIdentifier.PropMaxApduLengthAccepted, nData:=SIZEOF(nMaxApduSize), pData:=ADR(nMaxApduSize), bExecute:=TRUE);
			END_IF
			fbReadFifo.ProcessReadFifo();				
		E_BACnetRM_ClientState.eCalcAuto:
			IF nReadList>0 OR nWriteList>0 THEN
				IF eReadMode = E_BACnet_CommMode.eAuto THEN
					IF nMaxApduSize <= 480 THEN
						// [MS/TP Device]
						// > starting at 5 requests use RPM instead COV:
						_nRpmTreshold := 5;
						IF nMaxApduSize <= 206 THEN
							// For very small devices put only 10 properties into 1 request (prevent segmentation)
							nRPMPropertiesPerRequest := 10;
						ELSE
							nRPMPropertiesPerRequest := 20; 
						END_IF
					ELSE
						// [IP Device]
						// > Use more parallel requests
						nMaxParallelRequests := 50;
						_nRpmTreshold := 300;
					END_IF
					
					IF nReadList > _nRpmTreshold AND stSupportedServices.bSuppReadPropertyMultiple THEN
						eReadMode := E_BACnet_CommMode.eRpm;
					ELSIF stSupportedServices.bSuppSubscribeCOV THEN
						eReadMode := E_BACnet_CommMode.eCov;
					ELSIF stSupportedServices.bSuppReadPropertyMultiple THEN
						eReadMode := E_BACnet_CommMode.eRpm;
					ELSE
						eReadMode := E_BACnet_CommMode.eRp;
					END_IF
					bSuppRpm  := stSupportedServices.bSuppReadPropertyMultiple;
					bSuppCov  := stSupportedServices.bSuppSubscribeCov;
					bSuppCovP := stSupportedServices.bSuppSubscribeCOVProperty; 
				END_IF
				State:=E_BACnetRM_ClientState.eCreateRequests;
			ELSE
				State:=E_BACnetRM_ClientState.eCycle;
			END_IF
			State:=E_BACnetRM_ClientState.eCreateRequests;
		E_BACnetRM_ClientState.eCreateRequests:
			IF eReadMode = E_BACnet_CommMode.eAuto OR eReadMode = E_BACnet_CommMode.eRpm THEN
				fbReadFifo.bRpm:=stSupportedServices.bSuppReadPropertyMultiple;
			END_IF
			IF CreateReqList() THEN
				bUpdateReqs := FALSE;
				State:=E_BACnetRM_ClientState.eCycle;
			END_IF
		E_BACnetRM_ClientState.eCycle:
			IF bUpdateReqs THEN
				State:=E_BACnetRM_ClientState.eReInit;
				bUpdateReqs := FALSE;
				bReady:=FALSE;
			ELSE
				bReady:=TRUE;
				
				// Work on acyclic / dynamic requests:
				fbReadFifo.ProcessReadFifo();
				fbWriteFifo.ProcessWriteFifo();
				
				// Work on cyclic requests:
				IF stReqList <> 0 THEN
					_n := 0;
					WHILE nOpenReq < nMaxParallelRequests AND _n<nReqList DO								
						IF stReqList[nCurReq].pPtr <> 0 AND_THEN stReqList[nCurReq].fbBase^.IsReady() THEN
							IF stReqList[nCurReq].fbBase^.Send() THEN
								nOpenReq:=nOpenReq+1;
								IF nCurReq = 0 THEN
									IF _tCycleStartTime <> T#0S THEN
										diagCycleDuration:= TIME() - _tCycleStartTime;
									END_IF
									_tCycleStartTime := TIME();
								END_IF
							END_IF
						END_IF
						_n:=_n+1;
						nCurReq:=(nCurReq+1) MOD nReqList;
					END_WHILE
				END_IF
			END_IF
			IF NOT bConnected THEN
				State:=E_BACnetRM_ClientState.eReInit;
			END_IF
		E_BACnetRM_ClientState.eReInit:
			DeleteReqList();
			State:=E_BACnetRM_ClientState.eInit;
		E_BACnetRM_ClientState.eError:
			IF ((TIME()-_tReInitTime) > T#5S) THEN
				State:=E_BACnetRM_ClientState.eReInit;
			END_IF
	END_CASE
END_IF

{attribute 'hide'}
METHOD OnCOV
VAR_INPUT
	ePropID		: E_BACnetPropIdentifier;
END_VAR
END_METHOD

{attribute 'hide'}
METHOD OnReqError
VAR_INPUT
	iRequest		: I_BACnetRM_BaseReq;
	stResult		: POINTER TO SendDataRequestResult;
	sLogCode		: STRING			:= '';
END_VAR
VAR
	nLogType		: DWORD;
END_VAR
END_METHOD

METHOD INTERNAL OnRequestComplete
IF nOpenReq > 0 THEN
	nOpenReq:=nOpenReq-1;
END_IF
END_METHOD

METHOD INTERNAL AddReadEntry : BOOL
VAR_INPUT
	iObject 	: I_BACnetRM_BaseObject;
	ePropID 	: E_BACnetPropIdentifier;
	ePriority	: E_BACnet_Priority := E_BACnet_Priority.Invalid;
END_VAR
VAR_OUTPUT
	stResult	: POINTER TO ST_BACnetRM_ReadEntry;
END_VAR
VAR
	nTmp		: UDINT;
	nTmpSize	: UDINT;
	pTmp		: PVOID;
END_VAR
// Search for existing entry:
FOR nTmp := nReadList TO 1 BY -1 DO
	stResult := ADR(stReadList[nTmp-1]);
	IF (stResult^.iObject = iObject) AND_THEN (stResult^.ePropID = ePropID) THEN
		F_BA_LogMessage1(ADSLOG_MSGTYPE_ERROR, 'ARE05', 'Failed to initialize duplicate RemoteRead-Entry for Property "%d"!', F_INT(ePropID));
		RETURN;
	END_IF
END_FOR

IF (nReadList+1 >= nReadMax) THEN
	// Append list:
	nTmp := nReadMax+10;
	nTmpSize := nTmp*SIZEOF(ST_BACnetRM_ReadEntry);
	pTmp := __NEW(BYTE,nTmpSize);
	IF pTmp = 0 THEN
		RETURN;
	END_IF
	IF stReadList <> 0 THEN
		MEMCPY(pTmp, stReadList, nReadMax*SIZEOF(ST_BACnetRM_ReadEntry));
		__DELETE(stReadList);
	END_IF
	stReadList:=pTmp;
	nReadMax:=nTmp;
END_IF

// Create new entry:
stResult := ADR(stReadList[nReadList]);
nReadList := (nReadList+1);

// Initialize entry:
MEMSET(stResult, 0, SIZEOF(ST_BACnetRM_ReadEntry));
stResult^.iObject := iObject;
stResult^.ePropID := ePropID;
stResult^.nIndex := 16#FFFFFFFF;

AddReadEntry:=TRUE;
END_METHOD

METHOD INTERNAL AddWriteEntry : BOOL
VAR_INPUT
	iObject 	: I_BACnetRM_BaseObject;
	ePropID 	: E_BACnetPropIdentifier;
	ePriority	: E_BACnet_Priority := E_BACnet_Priority.Invalid;
END_VAR
VAR_OUTPUT
	stResult	: POINTER TO ST_BACnetRM_WriteEntry;
END_VAR
VAR
	nTmp		: UDINT;
	nTmpSize	: UDINT;
	pTmp		: PVOID;
END_VAR
// Search for existing entry:
FOR nTmp := nWriteList TO 1 BY -1 DO
	stResult := ADR(stWriteList[nTmp-1]);
	IF (stResult^.iObject = iObject) AND_THEN (stResult^.ePropID = ePropID) THEN
		IF (ePropID = E_BACnetPropIdentifier.PropPresentValue) AND_THEN (stResult^.nPriority <> TO_UDINT(ePriority)) THEN
			; // Allow requests on different priorities.
		ELSE
			F_BA_LogMessage1(ADSLOG_MSGTYPE_ERROR, 'AWE05', 'Failed to initialize duplicate RemoteWrite-Entry for Property "%d"!', F_INT(ePropID));
			RETURN;
		END_IF
	END_IF
END_FOR

IF (nWriteList+1 >= nWriteMax) THEN
	// Append list:
	nTmp := nWriteMax+10;
	nTmpSize := nTmp*SIZEOF(ST_BACnetRM_WriteEntry);
	pTmp := __NEW(BYTE,nTmpSize);
	IF pTmp = 0 THEN
		RETURN;
	END_IF
	IF stWriteList <> 0 THEN
		MEMCPY(pTmp, stWriteList, nWriteMax*SIZEOF(ST_BACnetRM_WriteEntry));
		__DELETE(stWriteList);
	END_IF
	stWriteList:=pTmp;
	nWriteMax:=nTmp;
END_IF

// Create new entry:
stResult := ADR(stWriteList[nWriteList]);
nWriteList := (nWriteList+1);

// Initialize entry:
MEMSET(stResult, 0, SIZEOF(ST_BACnetRM_WriteEntry));
stResult^.iObject := iObject;
stResult^.ePropID := ePropID;
stResult^.fCOVIncrement := 0.0;

AddWriteEntry := TRUE;
END_METHOD

METHOD INTERNAL AddFifoReadReq : BOOL
VAR_INPUT
	pReq : POINTER TO FB_BACnetRM_ReadProperty;
END_VAR
VAR
	entry : ST_BACnetRM_FifoEntry;
END_VAR
entry.fbRead:=pReq;
AddFifoReadReq:=fbReadFifo.AddFifoReq(entry);
END_METHOD

METHOD INTERNAL AddFifoWriteReq : BOOL
VAR_INPUT
	pReq : POINTER TO FB_BACnetRM_WriteProperty;
END_VAR
VAR
	entry : ST_BACnetRM_FifoEntry;
END_VAR
entry.fbWrite:=pReq;
AddFifoWriteReq:=fbWriteFifo.AddFifoReq(entry);
END_METHOD

{attribute 'hide'}
METHOD UpdateRequests 
VAR_INPUT
END_VAR
bUpdateReqs:=TRUE;
bReady:=FALSE;
END_METHOD

METHOD PRIVATE CreateReadReq : I_BACnetRM_BaseReq
VAR_INPUT
	eReadMode : E_BACnet_CommMode;
	stEntry : ST_BACnetRM_ReadEntry;
END_VAR
VAR
	stPtr : ST_BACnetRM_ReqPtr;
END_VAR
CASE eReadMode OF
	E_BACnet_CommMode.eCov:
		stPtr.fbCov:=__NEW(FB_BACnetRM_ReqCov);
		IF stPtr.fbCov <> 0 THEN
			stPtr.fbCov^(Client:=THIS^,iObject:=stEntry.iObject,  ePropID:=stEntry.ePropID, tLifetime:=tCOVLifeTime, pData:=stEntry.pData, nData:=stEntry.nData);
			stPtr.fbCov^.InitTimer();
		END_IF
		CreateReadReq:=stPtr.iReq;
		RETURN;
	E_BACnet_CommMode.eCovC:
		stPtr.fbCov:=__NEW(FB_BACnetRM_ReqCov);
		IF stPtr.fbCov <> 0 THEN
			stPtr.fbCov^(Client:=THIS^,iObject:=stEntry.iObject, bConfirmed:=TRUE, ePropID:=stEntry.ePropID, tLifetime:=tCOVLifeTime, pData:=stEntry.pData, nData:=stEntry.nData);
			stPtr.fbCov^.InitTimer();
		END_IF
		CreateReadReq:=stPtr.iReq;
		RETURN;
	E_BACnet_CommMode.eCovU:
		stPtr.fbCov:=__NEW(FB_BACnetRM_ReqCov);
		IF stPtr.fbCov <> 0 THEN
			stPtr.fbCov^(Client:=THIS^,iObject:=stEntry.iObject, bUnsubscribed:=TRUE, ePropID:=stEntry.ePropID, tLifetime:=tCOVLifeTime, pData:=stEntry.pData, nData:=stEntry.nData);
			stPtr.fbCov^.InitTimer();
		END_IF
		CreateReadReq:=stPtr.iReq;
		RETURN;
	E_BACnet_CommMode.eRp:
		stPtr.fbRead:=__NEW(FB_BACnetRM_ReqRead);
		IF stPtr.fbRead <> 0 THEN
			stPtr.fbRead^(Client:=THIS^,iObject:=stEntry.iObject, tCycleTime:=tReadCycleTime, ePropID:=stEntry.ePropID, pData:=stEntry.pData, nData:=stEntry.nData);
			stPtr.fbRead^.InitTimer();
		END_IF
		CreateReadReq:=stPtr.iReq;
		RETURN;
	E_BACnet_CommMode.eRpm:
		stPtr.fbRpm:=__NEW(FB_BACnetRM_ReqRpm);
		IF stPtr.fbRpm <> 0 THEN
			stPtr.fbRpm^(Client:=THIS^,iObject:=stEntry.iObject, tCycleTime:=tReadCycleTime);
			stPtr.fbRpm^.InitTimer();
		END_IF
		CreateReadReq:=stPtr.iReq;
		RETURN;
END_CASE
END_METHOD

METHOD PRIVATE CreateReqList : BOOL
VAR_INPUT
END_VAR
VAR
	i : UDINT;
	n : UDINT;
	nRpmEntries : UDINT;
	nReqs : UDINT;
	stPtr : ST_BACnetRM_ReqPtr;
	nReqsLeft : UDINT;
	pCurRpmReq : POINTER TO FB_BACnetRM_ReqRpm;
	bOptimizeCov : BOOL;
	nSize : UDINT;
END_VAR
DeleteReqList();

IF nReadList = 0 THEN
	CreateReqList:=TRUE;
	RETURN;
END_IF

// Calculate effective access mode and count RPM entries
FOR i:=0 TO nReadList-1 DO
	IF stReadList[i].iObject.ReadMode = E_BACnet_CommMode.eAuto THEN
		stReadList[i].eReadMode := eReadMode;
	ELSE
		stReadList[i].eReadMode := stReadList[i].iObject.ReadMode;
	END_IF
	IF F_IsCovReadMode(stReadList[i].eReadMode) THEN
		IF NOT bSuppCovP THEN
			IF NOT F_IsCovProperty(stReadList[i].iObject.ObjectType, stReadList[i].ePropID) THEN
				// ggf. error message if stReadList[i].fCOVIncrement <> 0.0
				IF bSuppRpm THEN
					stReadList[i].eReadMode := E_BACnet_CommMode.eRpm;
				ELSE
					stReadList[i].eReadMode := E_BACnet_CommMode.eRp;
				END_IF
			END_IF
		END_IF
		IF NOT bSuppCov THEN
			// ggf. error message that COV is configured but not available
			IF bSuppRpm THEN
				stReadList[i].eReadMode := E_BACnet_CommMode.eRpm;
			ELSE
				stReadList[i].eReadMode := E_BACnet_CommMode.eRp;
			END_IF
		END_IF
	END_IF
	IF stReadList[i].eReadMode = E_BACnet_CommMode.eRpm THEN
		nRpmEntries:=nRpmEntries+1;
	END_IF
END_FOR

// Calculate RPM request count
IF nRpmEntries > 0 THEN
	nReqs:=((nRpmEntries+nRPMPropertiesPerRequest-1)/nRPMPropertiesPerRequest);
END_IF

// Add single read requests + write repuests
nReqs := nReqs + (nReadList-nRpmEntries) + nWriteList;

stReqList:=__NEW(POINTER TO ST_BACnetRM_ReqPtr, nReqs);

IF stReqList = 0 THEN
	RETURN;
END_IF

FOR i:=0 TO nReadList-1 DO
	IF stReadList[i].eReadMode = E_BACnet_CommMode.eRpm THEN
		IF pCurRpmReq = 0 OR_ELSE pCurRpmReq^.nEntries = nRPMPropertiesPerRequest THEN
			stPtr.fbRpm:=__NEW(FB_BACnetRM_ReqRpm);
			IF stPtr.fbRpm = 0 THEN
				RETURN;
			END_IF
			nSize:=nRPMPropertiesPerRequest*SIZEOF(ST_BACnetRM_ReadEntry);
			stPtr.fbRpm^.pEntries:=__NEW(BYTE,nSize);
			IF stPtr.fbRpm^.pEntries = 0 THEN
				RETURN;
			END_IF
			IF pCurRpmReq <> 0 THEN
				pCurRpmReq^.InitTimer();
		 		pCurRpmReq^.UpdateRequest();		
			END_IF
			stPtr.fbRpm^.bFreeEntries:=TRUE;
			pCurRpmReq:=stPtr.fbRpm; 
			stPtr.fbRpm^(Client:=THIS^, iObject:=stReadList[i].iObject, tCycleTime:=tReadCycleTime);
			stReqList[nReqList]:=stPtr;		
	 		nReqList:=nReqList+1;
		END_IF 
		pCurRpmReq^.pEntries[pCurRpmReq^.nEntries]:=stReadList[i];
 		pCurRpmReq^.nEntries := pCurRpmReq^.nEntries + 1;	
	ELSE	
		stReqList[nReqList].iReq := CreateReadReq(stReadList[i].eReadMode, stReadList[i]);
		IF stReqList[nReqList].pPtr = 0 THEN
			RETURN;
		END_IF
		IF F_IsCovReadMode(stReadList[i].eReadMode) THEN
			bOptimizeCov := TRUE;
		END_IF
		nReqList:=nReqList+1;
	END_IF
END_FOR

IF pCurRpmReq <> 0 THEN
	stPtr.fbRpm^.InitTimer();
	stPtr.fbRpm^.UpdateRequest();
END_IF

IF bOptimizeCov THEN
	OptimizeCOV();
END_IF

IF (nWriteList > 0) THEN
	FOR i:=0 TO nWriteList-1 DO
		stReqList[nReqList].fbWrite := __NEW(FB_BACnetRM_ReqWrite);
		IF stReqList[nReqList].pPtr = 0 THEN
			RETURN;
		END_IF	
		stReqList[nReqList].fbWrite^(Client:=THIS^, iObject:=stWriteList[i].iObject, ePropID:=stWriteList[i].ePropID, tCycleTime:=tWriteCycleTime, pData:=stWriteList[i].pData, nData:=stWriteList[i].nData, pEnable:=stWriteList[i].pEnable, pNull:=stWriteList[i].pNull, fCOVIncrement:=stWriteList[i].fCOVIncrement, ePriority:=TO_INT(stWriteList[i].nPriority));
		stReqList[nReqList].fbWrite^.InitTimer();
		nReqList:=nReqList+1;
	END_FOR
END_IF

nCurReq := 0;
nOpenReq := 0;
CreateReqList:=TRUE;
END_METHOD

METHOD PRIVATE DeleteReqList
VAR_INPUT
END_VAR
VAR
	i : UDINT;
END_VAR
IF nReqList > 0 AND stReqList <> 0 THEN
	FOR i:=0 TO nReqList-1 DO
		IF stReqList[i].nByte <> 0 THEN
			CASE stReqList[i].iReq.GetRequestType() OF
				E_BACnetRM_RequestType.eRead:__DELETE(stReqList[i].fbRead);
				E_BACnetRM_RequestType.eReadPropertyMultiple:__DELETE(stReqList[i].fbRpm); 
				E_BACnetRM_RequestType.eWrite:__DELETE(stReqList[i].fbWrite);
				E_BACnetRM_RequestType.eWritePropertyMultiple:__DELETE(stReqList[i].fbWpm);
				E_BACnetRM_RequestType.eCOV_C:__DELETE(stReqList[i].fbCov);
				E_BACnetRM_RequestType.eCOV:__DELETE(stReqList[i].fbCov);
				E_BACnetRM_RequestType.eCOV_U:__DELETE(stReqList[i].fbCov);
			END_CASE
		END_IF
	END_FOR
	__DELETE(stReqList);
	stReqList:=0;
	nReqList:=0;
END_IF
END_METHOD

// Optimizes request count per object.
// > If a single object has more than one request, these multiple requests can be handled via a single RPM-request.
METHOD PRIVATE OptimizeCOV : BOOL
VAR
	i : UDINT;
	j : UDINT;
	bSkipCov : BOOL;
END_VAR
IF (nReqList > 0) THEN
	FOR i:=0 TO nReqList-1 DO
		IF stReqList[i].iReq <> 0 AND_THEN F_IsCovReqType(stReqList[i].iReq) AND_THEN stReqList[i].fbCov^.Master = 0 THEN
			bSkipCov := F_IsCovProperty(stReqList[i].fbCov^.iObject.ObjectType, stReqList[i].fbCov^.ePropID);
			FOR j:=i+1 TO nReqList-1 DO
				IF stReqList[j].iReq <> 0 AND_THEN F_IsCovReqType(stReqList[j].iReq) AND_THEN stReqList[i].fbCov^.iObject.ObjectID = stReqList[j].fbCov^.iObject.ObjectID THEN
					 stReqList[i].fbCov^.AddCovSlave(stReqList[j].fbCov);
					 stReqList[j].fbCov^.Master:=stReqList[i].fbCov;
					 IF stReqList[j].fbCov^.fCOVIncrement = 0 AND F_IsCovProperty(stReqList[j].fbCov^.iObject.ObjectType, stReqList[j].fbCov^.ePropID) THEN
						 IF bSkipCov THEN
						 	stReqList[j].fbCov^.SendSubscription:=FALSE;
						 ELSE
							 bSkipCov:=TRUE;
						 END_IF
					 END_IF
				END_IF
			END_FOR
		END_IF
	END_FOR
END_IF
END_METHOD

// Called after online change.
{attribute 'call_after_online_change_slot' := '10'}
METHOD PROTECTED OnPostOnlineChange
IF iServer <> 0 THEN
	FW_SafeRelease(ADR(iServer));
	iServer:=0;
END_IF
IF iClient <> 0 THEN
	FW_SafeRelease(ADR(iClient));
	iClient:=0;
END_IF
iDevice:=0;

State:=E_BACnetRM_ClientState.eReInit;
END_METHOD

PROPERTY Error : BOOL
GET
Error := (eErrorID <> E_BACnet_Error.eNoError);
END_GET
END_PROPERTY

PROPERTY ObjectID : T_BACnet_ObjectIdentifier
GET
ObjectID := tObjectID;
END_GET
END_PROPERTY

PROPERTY ObjectInstance : UDINT
GET
ObjectInstance := nDeviceInstance;
END_GET
END_PROPERTY

PROPERTY ObjectType : E_BACnetObjType
GET
ObjectType := E_BACnetObjType.ObjDevice;
END_GET
END_PROPERTY

PROPERTY OpenRequestCount : UDINT
GET
OpenRequestCount:=nOpenReq;
END_GET
SET
nOpenReq:=OpenRequestCount;
END_SET
END_PROPERTY

PROPERTY ReadMode : E_BACnet_CommMode
GET
ReadMode:=eReadMode;
END_GET
SET
eReadMode:=ReadMode;
END_SET
END_PROPERTY

PROPERTY Ready : BOOL
GET
Ready := bReady;
END_GET
END_PROPERTY

PROPERTY State : E_BACnetRM_ClientState
GET
State := eState;
END_GET
SET
PRIVATE 
VAR
END_VAR
IF (State = E_BACnetRM_ClientState.eError) THEN
	_tReInitTime := TIME();
END_IF

eState := State;
END_SET
END_PROPERTY

METHOD FB_Exit : BOOL
VAR_INPUT
	 bInCopyCode : BOOL; // if TRUE, the exit method is called for exiting an instance that is copied afterwards (online change).
END_VAR
IF iServer <> 0 THEN
	iServer.OnPlcAction(E_BACnet_PlcAction.eSuspend);
	iServer:=0;
END_IF
IF iClient <> 0 THEN
	FW_SafeRelease(ADR(iClient));
	iClient:=0;
END_IF

iDevice:=0;

DeleteReqList();

IF stReadList <> 0 THEN
	__DELETE(stReadList);
	stReadList:=0;
END_IF
IF stWriteList <> 0 THEN
	__DELETE(stWriteList);
	stWriteList:=0;
END_IF
END_METHOD

END_FUNCTION_BLOCK

// POUs/Remote/Requests/[Internal]/FB_BACnetRM_ReqFifo
{attribute 'c++_compatible'}
{attribute 'enable_dynamic_creation'}
{attribute 'hide'}
FUNCTION_BLOCK FB_BACnetRM_ReqFifo EXTENDS FB_BACnetRM_ReqBase
VAR_INPUT
	bRpm : BOOL;
	bWpm : BOOL;
END_VAR
VAR
	pReqFifo	: POINTER TO ST_BACnetRM_FifoEntry;
	nReqFifo	: UDINT := 0;
	nMaxFifo	: UDINT := 0;
	nPendFifo	: UDINT := 0;
END_VAR

METHOD INTERNAL AddFifoReq : BOOL
VAR_INPUT
	pEntry : ST_BACnetRM_FifoEntry;
END_VAR
VAR
	nTmp : UDINT;
	nTmpSize : UDINT;
	pTmp : POINTER TO ST_BACnetRM_FifoEntry;
END_VAR
IF nReqFifo+1 >= nMaxFifo THEN
	nTmp := 2*nMaxFifo+100;
	nTmpSize := nTmp*SIZEOF(ST_BACnetRM_FifoEntry);
	pTmp := __NEW(BYTE,nTmpSize);
	IF pTmp = 0 THEN
		RETURN;
	END_IF
	IF pReqFifo <> 0 THEN
		MEMCPY(pTmp, pReqFifo, nMaxFifo*SIZEOF(ST_BACnetRM_FifoEntry));
		__DELETE(pReqFifo);
	END_IF
	pReqFifo:=pTmp;
	nMaxFifo:=nTmp;
END_IF

pReqFifo[nReqFifo]:=pEntry;
nReqFifo:=nReqFifo+1;

AddFifoReq:=TRUE;
END_METHOD

METHOD INTERNAL ProcessReadFifo : BOOL
VAR_INPUT
END_VAR
VAR
	pRequest : ST_BACnetRM_ReqPtr;
	nSize : UDINT;
	n :UDINT;
	pEntries : POINTER TO ST_BACnetRM_ReadEntry;	
	x : UDINT;
	iTmpFB : I_BACnetRM_BasicReq;
END_VAR
IF Valid THEN
	WHILE Client.nOpenReq < Client.nMaxParallelRequests AND nReqFifo > 0 DO		
		IF bRpm AND nReqFifo>1 THEN
			n:=0;
			nSize:=MIN(nReqFifo, Client.nRPMPropertiesPerRequest)*SIZEOF(ST_BACnetRM_ReadEntry);
			pRequest.fbRpm := __NEW(FB_BACnetRM_ReqRpm);
			IF pRequest.fbRpm = 0 THEN
				RETURN;
			END_IF
			pEntries:=__NEW(BYTE,nSize);
			IF pEntries = 0 THEN
				__DELETE(pRequest.fbRpm);
				RETURN;
			END_IF
			WHILE n<nReqFifo AND n < Client.nRPMPropertiesPerRequest DO
				pEntries[n].iObject:=pReqFifo[n].fbRead^.iObject;
				pEntries[n].ePropID:=pReqFifo[n].fbRead^.ePropID;
				pEntries[n].pData:=pReqFifo[n].fbRead^.pData;
				pEntries[n].nData:=pReqFifo[n].fbRead^.nData;
				pEntries[n].nIndex:=pReqFifo[n].fbRead^.nIndex;
				IF __QUERYINTERFACE(pReqFifo[0].fbRead^, iTmpFB) THEN
					pEntries[n].iReadFB:=iTmpFB;
				END_IF
				n:=n+1;
			END_WHILE		
			pRequest.fbRpm^(Client:=Client, iObject:=pReqFifo[0].fbRead^.iObject, pEntries:=pEntries, nEntries:=n, bFreeEntries:=TRUE);
			IF pRequest.fbRpm^.UpdateRequest() AND_THEN pRequest.fbRpm^.Send() THEN
				Client.OpenRequestCount:=Client.nOpenReq+1;
				pReqFifo[0].fbRead^.Request:=pRequest;
				pReqFifo[0].fbRead^.bReqRPM:=TRUE;
				IF nReqFifo-n > 0 THEN
					MEMMOVE(pReqFifo, ADR(pReqFifo[n]), (nReqFifo-n)*SIZEOF(ST_BACnetRM_ReadEntry));
				END_IF
				nReqFifo:=nReqFifo-n;
			ELSE
				__DELETE(pRequest.fbRpm);
				RETURN;
			END_IF
		ELSE
			pRequest.fbRead := __NEW(FB_BACnetRM_ReqRead);
			IF pRequest.fbRead = 0 THEN
				RETURN;
			END_IF
			__QUERYINTERFACE(pReqFifo[0].fbRead^, iTmpFB);
			pRequest.fbRead^(Client:=Client, iObject:=pReqFifo[0].fbRead^.iObject, pData:=pReqFifo[0].fbRead^.pData, nData:=pReqFifo[0].fbRead^.nData, ePropID:=pReqFifo[0].fbRead^.ePropID, iReadFB:=iTmpFB);
			Client.OpenRequestCount:=Client.nOpenReq+1;
			pReqFifo[0].fbRead^.Request:=pRequest;	
			pReqFifo[0].fbRead^.bReqRPM:=FALSE;
			IF pRequest.fbRead^.Send() THEN
				IF nReqFifo-n > 0 THEN
					MEMMOVE(pReqFifo, ADR(pReqFifo[1]),(nReqFifo-1)*SIZEOF(ST_BACnetRM_ReadEntry));
				END_IF
				nReqFifo:=nReqFifo-1;
			ELSE
				Client.OpenRequestCount:=Client.nOpenReq-1;
				__DELETE(pRequest.fbRead);
				RETURN;
			END_IF
		END_IF
	END_WHILE
	
	ProcessReadFifo:=TRUE;
ELSE
	// (BETA) ... Output Error
END_IF
END_METHOD

METHOD INTERNAL ProcessWriteFifo : BOOL
VAR_INPUT
END_VAR
VAR
	pRequest : ST_BACnetRM_ReqPtr;
	nSize : UDINT;
	n : UDINT;
	pEntries : POINTER TO ST_BACnetRM_WriteEntry;
	iTmpFB : I_BACnetRM_BasicReq;
END_VAR
IF Valid THEN
	WHILE Client.nOpenReq < Client.nMaxParallelRequests AND nReqFifo > 0 DO		
		IF bWpm THEN
			n:=0;
			nSize:=MIN(nReqFifo, Client.nRPMPropertiesPerRequest)*SIZEOF(ST_BACnetRM_WriteEntry);
			pRequest.fbWpm:= __NEW(FB_BACnetRM_ReqWpm);
			IF pRequest.fbWpm = 0 THEN
				RETURN;
			END_IF
			pEntries:=__NEW(BYTE,nSize);
			IF pEntries = 0 THEN
				__DELETE(pRequest.fbWpm);
				RETURN;
			END_IF
			WHILE n<nReqFifo-1 AND n < Client.nRPMPropertiesPerRequest DO
				pEntries[n].iObject:=pReqFifo[n].fbWrite^.iObject;
				pEntries[n].ePropID:=pReqFifo[n].fbWrite^.ePropID;
				pEntries[n].pData:=pReqFifo[n].fbWrite^.pData;
				pEntries[n].nData:=pReqFifo[n].fbWrite^.nData;
				pEntries[n].nIndex:=pReqFifo[n].fbWrite^.nIndex;
				IF __QUERYINTERFACE(pReqFifo[0].fbWrite^, iTmpFB) THEN
					pEntries[n].iWriteFB:=iTmpFB;
				END_IF
				n:=n+1;
			END_WHILE
			pRequest.fbWpm^(Client:=Client, pEntries:=pEntries, nEntries:=n, bFreeEntries:=TRUE);
			IF pRequest.fbWpm^.UpdateRequest() AND_THEN pRequest.fbWpm^.Send() THEN
				Client.OpenRequestCount:=Client.nOpenReq+1;
				pReqFifo[0].fbRead^.Request:=pRequest;
				pReqFifo[0].fbWrite^.bRequestWPM:=TRUE;
				IF nReqFifo-n > 0 THEN
					MEMMOVE(pReqFifo, ADR(pReqFifo[n]), (nReqFifo-n)*SIZEOF(ST_BACnetRM_WriteEntry));
				END_IF
				nReqFifo:=nReqFifo-n;
			ELSE
				__DELETE(pRequest.fbWpm);
				RETURN;
			END_IF
		ELSE
			pRequest.fbWrite := __NEW(FB_BACnetRM_ReqWrite);
			IF pRequest.fbWrite = 0 THEN
				RETURN;
			END_IF
			pRequest.fbWrite^.pData:=pReqFifo[0].fbWrite^.pData;
			pRequest.fbWrite^.nData:=pReqFifo[0].fbWrite^.nData;
			__QUERYINTERFACE(pReqFifo[0].fbWrite^, iTmpFB);
			pRequest.fbWrite^(Client:=Client, iObject:=pReqFifo[0].fbWrite^.iObject, ePropID:=pReqFifo[0].fbWrite^.ePropID, iWriteFB:=iTmpFB);
			IF pRequest.fbWrite^.Send() THEN
				pReqFifo[0].fbWrite^.Request:=pRequest;	
				pReqFifo[0].fbWrite^.bRequestWPM:=FALSE;
				Client.OpenRequestCount:=Client.nOpenReq+1;
				IF (nReqFifo-1) > 0 THEN
					MEMMOVE(pReqFifo, ADR(pReqFifo[1]),(nReqFifo-1)*SIZEOF(ST_BACnetRM_WriteEntry));
				END_IF
				nReqFifo:=nReqFifo-1;
			ELSE
				__DELETE(pRequest.fbWrite);
				RETURN;
			END_IF
		END_IF
	END_WHILE
	
	ProcessWriteFifo:=TRUE;
ELSE
	// (BETA) ... Output Error
END_IF
END_METHOD

PROPERTY Valid : BOOL
GET
// Hint:
// > Don't call "super()"!
//   The "iObject" Interface-pointer is ignored to this instance because it is unused.
Valid := (__ISVALIDREF(Client));
END_GET
END_PROPERTY

METHOD FB_Exit : BOOL
VAR_INPUT
	 bInCopyCode : BOOL; // if TRUE, the exit method is called for exiting an instance that is copied afterwards (online change).
END_VAR
IF pReqFifo <> 0 THEN
	__DELETE(pReqFifo);
	pReqFifo:=0;
END_IF
END_METHOD

END_FUNCTION_BLOCK

// POUs/Remote/Requests/[Internal]/[Base]/FB_BACnetRM_ReqBase
{attribute 'c++_compatible'}
{attribute 'enable_dynamic_creation'}
{attribute 'hide'}
FUNCTION_BLOCK FB_BACnetRM_ReqBase IMPLEMENTS I_BACnetRM_BaseReq
VAR_INPUT
	{attribute 'initialize_on_call'}
	{attribute 'no_copy'}
	Client : REFERENCE TO FB_BACnet_Client;
	iObject : I_BACnetRM_BaseObject;
END_VAR

METHOD PROTECTED OnError
VAR_INPUT
	stResult		: POINTER TO SendDataRequestResult;
	sLogCode		: STRING			:= '';
END_VAR
VAR
	i : UDINT;
END_VAR
IF (iObject <> 0) THEN
	iObject.OnReqError(THIS^, stResult, 'OE01');
END_IF
END_METHOD

PROPERTY Valid : BOOL
GET
VAR
	iTest : BOOL;
END_VAR
Valid := (__ISVALIDREF(Client)) AND (iObject <> 0);
END_GET
END_PROPERTY

METHOD GetRequestType : E_BACnetRM_RequestType
VAR_INPUT
END_VAR
GetRequestType:=E_BACnetRM_RequestType.eUndefined;
END_METHOD

METHOD IsReady : BOOL
END_METHOD

METHOD Send : BOOL
VAR
	_ClTmp : ITcIoBACnetPlcClient;
END_VAR
END_METHOD

END_FUNCTION_BLOCK

// POUs/Remote/Requests/[Internal]/FB_BACnetRM_ReqRpm
{attribute 'c++_compatible'}
{attribute 'enable_dynamic_creation'}
{attribute 'hide'}
FUNCTION_BLOCK FB_BACnetRM_ReqRpm EXTENDS FB_BACnetRM_ReqBasic
VAR_INPUT
	pEntries : POINTER TO ST_BACnetRM_ReadEntry;
	nEntries : UDINT;
	bFreeEntries : BOOL; 
END_VAR
VAR_OUTPUT
	bInit : BOOL;
END_VAR
VAR 
	req : SendDataRequest;
	pTmp : POINTER TO ST_BACnetRM_RpmListEntry;
END_VAR

IF NOT __ISVALIDREF(Client) THEN
	bError:=TRUE;
END_IF

SUPER^();

{attribute 'hide'}
METHOD Send : BOOL
IF Valid THEN
	IF stReq = 0 THEN
		RETURN;
	END_IF
	
	Send:=SUPER^.Send();
END_IF
END_METHOD

METHOD INTERNAL UpdateRequest : BOOL
VAR_INPUT
END_VAR
VAR
	nSize : UDINT;
	i : UDINT;
	nTmpSize : UDINT;
END_VAR
IF Valid THEN
	IF stReq <> 0 AND_THEN stReq^.pData <> 0 THEN
		pTmp:=stReq^.pData;
		__DELETE(pTmp);
		stReq^.pData:=0;
	END_IF
	nTmpSize := SIZEOF(ST_BACnetRM_RpmListEntry)*nEntries;
	pTmp := __NEW(BYTE,nTmpSize);
	IF pTmp = 0 THEN
		RETURN;
	END_IF
	
	FOR i:=0 TO nEntries-1 DO
		pTmp[i].tObjectID := pEntries[i].iObject.ObjectID;
		pTmp[i].ePropID := pEntries[i].ePropID;
		pTmp[i].nArrayIndex := 0;
		pTmp[i].nValidBits := 0;
		pTmp[i].nPriority := 0;
		pTmp[i].nEntrySize := SIZEOF(ST_BACnetRM_RpmListEntry) - 8;
		IF i <> nEntries -1 THEN
			pTmp[i].nEntrySize := pTmp[i].nEntrySize + 16#80000000;
		END_IF
	END_FOR
	
	stReq := ADR(req);
	stReq^.pData := pTmp;
	stReq^.nData := nTmpSize;
	
	stReq^.service := E_BACnetConfirmedService.SrvReadPropertyMultiple;
	stReq^.deviceId := Client.ObjectInstance;
	
	bInit:=TRUE;
	
	UpdateRequest:=TRUE;
ELSE
	// (BETA) ... Output Error
END_IF
END_METHOD

METHOD PRIVATE Free
VAR_INPUT
END_VAR
IF bFreeEntries AND pEntries <> 0 THEN
	__DELETE(pEntries);
	pEntries:=0;
	bFreeEntries:=FALSE;
END_IF

IF stReq <> 0 AND_THEN stReq^.pData <> 0 THEN
	pTmp:=req.pData;
	__DELETE(pTmp);
	req.pData:=0;
	stReq:=0;
END_IF
END_METHOD

METHOD PROTECTED OnError
VAR_INPUT
	stResult		: POINTER TO SendDataRequestResult;
	sLogCode		: STRING			:= '';
END_VAR
VAR
	i : UDINT;
END_VAR
// Do not call super! Handle each entry's error:
// SUPER^.OnError(eResult, sLogCode);

FOR i:=0 TO nEntries-1 DO
	IF pEntries[i].iReadFB <> 0 THEN
		pEntries[i].iReadFB.SetError();
		IF (pEntries[i].iObject <> 0) THEN
			pEntries[i].iObject.OnReqError(THIS^, stResult, 'OE07');
		END_IF	
	END_IF
END_FOR
END_METHOD

METHOD PROTECTED ProcessResult : HRESULT
VAR_INPUT
	pResult	: POINTER TO SendDataRequestResult;
END_VAR
VAR
	pPropList : POINTER TO ST_BACnetRM_RpmListEntry;
	i : UDINT;
END_VAR
IF pResult^.service <> E_BACnetConfirmedService.SrvReadPropertyMultiple THEN
	ProcessResult:=E_FAIL;
	RETURN;
END_IF

IF pEntries = 0 THEN // Request object has already been deleted
	ProcessResult:=E_FAIL;
	RETURN;
END_IF

// set all entries to error, all good entries in response will be set to good afterwards
FOR i:=0 TO nEntries-1 DO
	IF pEntries[i].iReadFB <> 0 THEN
		pEntries[i].iReadFB.SetError();
	END_IF
	
	pEntries[i]._bError := TRUE;
END_FOR

// copy data:
pPropList := pResult^.pData;
WHILE pPropList <> 0 DO
	_WritePropEntry(pPropList);
	pPropList := F_BACnet_NextListElem(pPropList, pPropList^.nEntrySize);
END_WHILE

// Evaluate remaining errors:
FOR i:=0 TO nEntries-1 DO
	IF (pEntries[i]._bError) AND_THEN (pEntries[i].iObject <> 0) THEN
		pEntries[i].iObject.OnReqError(THIS^, pResult, 'OE28');
	END_IF
END_FOR

ProcessResult:=S_OK;
END_METHOD

METHOD GetRequestType : E_BACnetRM_RequestType
VAR_INPUT
END_VAR
GetRequestType := E_BACnetRM_RequestType.eReadPropertyMultiple;
END_METHOD

METHOD PRIVATE _WritePropEntry : BOOL
VAR_INPUT
	pEntry : POINTER TO ST_BACnetRM_RpmListEntry;
END_VAR
VAR
	i : UDINT;
END_VAR
FOR i:=0 TO nEntries-1 DO
	IF (pEntries[i].iObject.ObjectID = pEntry^.tObjectID) AND (pEntries[i].ePropID = pEntry^.ePropID) THEN
		CopyRemoteData(pEntries[i].iObject, pEntry^.ePropID ,pEntries[i].pData, pEntries[i].nData, F_BACnet_EndOf(pEntry, SIZEOF(ST_BACnetRM_RpmListEntry)), F_BACnet_ElemSize(pEntry^.nEntrySize)-16); 
		IF pEntries[i].iReadFB <> 0 THEN
			pEntries[i].iReadFB.SetReady();
		END_IF
		pEntries[i]._bError := FALSE;
		
		_WritePropEntry:=TRUE;
	END_IF
END_FOR
END_METHOD

METHOD FB_exit : BOOL
VAR_INPUT
	bInCopyCode : BOOL; // if TRUE, the exit method is called for exiting an instance that is copied afterwards (online change).
END_VAR
Free();
END_METHOD

END_FUNCTION_BLOCK

// POUs/Remote/Requests/[Internal]/[Base]/FB_BACnetRM_ReqBasic
{attribute 'c++_compatible'}
{attribute 'enable_dynamic_creation'}
{attribute 'hide'}
FUNCTION_BLOCK FB_BACnetRM_ReqBasic EXTENDS FB_BACnetRM_ReqBase IMPLEMENTS ITcIoBACnetServiceResponseSink
VAR_INPUT
	tCycleTime : TIME := T#5S;
END_VAR
VAR_OUTPUT
	bBusy : BOOL;
	bError : BOOL;
	bReady : BOOL;
END_VAR
VAR
	{attribute 'hide'}
	stReq : POINTER TO SendDataRequest;
	timer : TON;
END_VAR

{attribute 'c++_compatible'}
{attribute 'minimal_input_size' := '4'}
{attribute 'pack_mode' := '4'}
{attribute 'hide'}
METHOD OnSendPropertyDataRequest : HRESULT
VAR_INPUT
	pResult	: POINTER TO SendDataRequestResult;
END_VAR
IF (Valid) AND_THEN (pResult <> 0) THEN
	IF F_BACnetRM_IsErrorSet(pResult) THEN
		SetError();
		OnError(pResult, 'OSPDR04');
		OnSendPropertyDataRequest:=S_FALSE;
	ELSE
		IF S_OK = ProcessResult(pResult) THEN
			SetReady();
			OnSendPropertyDataRequest:=S_OK;
		ELSE
			OnSendPropertyDataRequest:=S_FALSE;
		END_IF	
	END_IF
	Client.OnRequestComplete();
END_IF
END_METHOD

METHOD INTERNAL InitTimer : BOOL
VAR_INPUT
END_VAR
timer(IN:=FALSE, PT:=T#1MS);
timer(IN:=TRUE, PT:=T#1MS);
END_METHOD

{attribute 'hide'}
METHOD SetBusy
bBusy := TRUE;
bError := FALSE;
bReady := FALSE;
END_METHOD

{attribute 'hide'}
METHOD SetError
bBusy := FALSE;
bError := TRUE;
bReady := FALSE;
END_METHOD

{attribute 'hide'}
METHOD SetReady
bBusy := FALSE;
bError := FALSE;
bReady := TRUE;
END_METHOD

{attribute 'c++_compatible'}
{attribute 'minimal_input_size' := '4'}
{attribute 'pack_mode' := '4'}
{attribute 'hide'}
METHOD TcAddRef : UDINT
END_METHOD

{attribute 'c++_compatible'}
{attribute 'minimal_input_size' := '4'}
{attribute 'pack_mode' := '4'}
{attribute 'hide'}
METHOD TcQueryInterface : HRESULT
VAR_INPUT
	iid	: REFERENCE TO IID;
	pipItf	: POINTER TO PVOID;
END_VAR
VAR
	ipSink : ITcIoBACnetServiceResponseSink;
	ipUnknown : ITcUnknown;	
END_VAR
IF GuidsEqual(ADR(iid), ADR(TC_GLOBAL_IID_LIST.IID_ITcIoBACnetServiceResponseSink)) THEN
	ipSink := THIS^; // cast to interface pointer
	pipItf^ := ITCUNKNOWN_TO_PVOID(ipSink);
	TcAddRef();
	TcQueryInterface := S_OK;
ELSIF GuidsEqual(ADR(iid), ADR(TC_GLOBAL_IID_LIST.IID_ITcUnknown)) THEN
	ipUnknown := THIS^; // cast to interface pointer
	pipItf^ := ITCUNKNOWN_TO_PVOID(ipUnknown);
	TcAddRef();
	TcQueryInterface := S_OK;
ELSE
	TcQueryInterface := E_HRESULTAdsErr.NOINTERFACE ; //Call super if this fb extends some other
END_IF
END_METHOD

{attribute 'c++_compatible'}
{attribute 'minimal_input_size' := '4'}
{attribute 'pack_mode' := '4'}
{attribute 'hide'}
METHOD TcRelease : UDINT
END_METHOD

METHOD PROTECTED CopyRemoteData : BOOL
VAR_INPUT
	iObject : I_BACnetRM_BaseObject;
	ePropID : E_BACnetPropIdentifier;
	pDst : PVOID;
	nDst : UDINT;
	pRead : PVOID;
	nRead : UDINT;
END_VAR
VAR
	i 	 : INT;
	pByte : POINTER TO BYTE;
	pSchedPv : POINTER TO ST_BACnet_ValueList;
END_VAR
// Individual treatment:
CASE (ePropID) OF
	E_BACnetPropIdentifier.PropPresentValue:
		IF iObject.ObjectType = E_BACnetObjType.ObjSchedule THEN
			IF (nRead >= 16) THEN
				pSchedPv := pRead;
				CASE pSchedPv^.listEntry.eValueChoice OF
					E_BACnet_ValueChoice.eBoolValue:
						MEMCPY(pDst, ADR(pSchedPv^.listEntry.stValue), MIN(SIZEOF(BOOL),nDst)); 
					E_BACnet_ValueChoice.eRealValue:
						MEMCPY(pDst, ADR(pSchedPv^.listEntry.stValue), MIN(SIZEOF(REAL),nDst)); 
					E_BACnet_ValueChoice.eUnsignedValue:
						MEMCPY(pDst, ADR(pSchedPv^.listEntry.stValue), MIN(SIZEOF(UDINT),nDst)); 
					E_BACnet_ValueChoice.eEnumerationValue:
						MEMCPY(pDst, ADR(pSchedPv^.listEntry.stValue.nEnumValue), MIN(SIZEOF(UDINT),nDst)); 
				END_CASE
			
				CopyRemoteData := TRUE;
			END_IF
		END_IF
		
	// Consider enumerations with smaller base-types:
	E_BACnetPropIdentifier.PropCurrentlyActivePriority:
		nRead := nDst;
		
END_CASE

// Check if received bytes match expected size:
IF (NOT CopyRemoteData) AND_THEN (nRead <= nDst) THEN
	// Individual treatment:
	CASE (ePropID) OF
		E_BACnetPropIdentifier.PropStatusFlags:
			pByte:=pDst;
			FOR i:=0 TO 3 DO
				IF F_BACnet_IsBitFieldBitSetPtr(pRead, i) THEN
					pByte[i]:=1;
				ELSE
					pByte[i]:=0;
				END_IF
			END_FOR
			
		E_BACnetPropIdentifier.PropAckedTransitions,
		E_BACnetPropIdentifier.PropEventEnable:
			pByte:=pDst;
			FOR i:=0 TO 2 DO
				IF F_BACnet_IsBitFieldBitSetPtr(pRead, i) THEN
					pByte[i]:=1;
				ELSE
					pByte[i]:=0;
				END_IF
			END_FOR
			
	ELSE
		// Default treatment:
		MEMCPY(pDst, pRead, MIN(nRead,nDst)); 
	END_CASE
	
	CopyRemoteData := TRUE;
END_IF

IF (CopyRemoteData) THEN
	// Notify object about changed value:
	iObject.OnCOV(ePropID);
ELSE
	F_BA_LogMessage3(ADSLOG_MSGTYPE_ERROR, 'CRD51', 'Unable to process remote data due to invalid size (Property: "%d", Read: %d Bytes, Expected: %d Bytes)!', F_INT(ePropID), F_UDINT(nRead), F_UDINT(nDst));
END_IF
END_METHOD

METHOD PROTECTED ProcessResult : HRESULT
VAR_INPUT
	pResult	: POINTER TO SendDataRequestResult;
END_VAR
ProcessResult:=S_OK;
END_METHOD

METHOD Send : BOOL
VAR
	_ClTmp : ITcIoBACnetPlcClient;
END_VAR
IF Valid THEN
	_ClTmp := Client.iClient;
	
	SetBusy();
	IF S_OK = _ClTmp.SendPropertyDataRequest(stReq, THIS^) THEN
		Send:=TRUE;
		StartTimer();
	ELSE
		SetError();
		Send:=FALSE; 
	END_IF
END_IF
END_METHOD

METHOD PROTECTED StartTimer : BOOL
VAR_INPUT
END_VAR
timer(IN:=FALSE, PT:=tCycleTime);
timer(IN:=TRUE, PT:=tCycleTime);
END_METHOD

METHOD GetRequestType : E_BACnetRM_RequestType
VAR_INPUT
END_VAR
GetRequestType:=E_BACnetRM_RequestType.eUndefined;
END_METHOD

METHOD IsReady : BOOL
VAR_INPUT
END_VAR
timer(Q=>IsReady);
IF bBusy THEN
	IsReady:=FALSE;
END_IF
END_METHOD

END_FUNCTION_BLOCK

// POUs/Remote/Requests/[Internal]/FB_BACnetRM_ReqRead
{attribute 'c++_compatible'}
{attribute 'enable_dynamic_creation'}
{attribute 'hide'}
FUNCTION_BLOCK FB_BACnetRM_ReqRead EXTENDS FB_BACnetRM_ReqBasic
VAR_INPUT
	ePropID : E_BACnetPropIdentifier;
	pData : PVOID;
	nData : UDINT;
	iReadFB : I_BACnetRM_BasicReq;
END_VAR
VAR 
	req : SendDataRequest;
END_VAR

IF NOT __ISVALIDREF(Client) THEN
	bError:=TRUE;
END_IF

SUPER^();

{attribute 'hide'}
METHOD Send : BOOL
IF Valid THEN
	IF stReq = 0 THEN
		IF ePropID = E_BACnetPropIdentifier.PropLogBuffer THEN
			req.service := E_BACnetConfirmedService.SrvReadRange;
		ELSE
			req.service := E_BACnetConfirmedService.SrvReadProperty;
		END_IF	
		req.objectIdentifier := iObject.ObjectID;
		req.propertyIdentifier := ePropID;
		req.pData := pData;
		req.nData := nData;
		req.deviceId := Client.ObjectInstance;
		stReq := ADR(req);
	END_IF
	
	Send:=SUPER^.Send();
END_IF
END_METHOD

METHOD PROTECTED OnError
VAR_INPUT
	stResult		: POINTER TO SendDataRequestResult;
	sLogCode		: STRING			:= '';
END_VAR
SUPER^.OnError(stResult, sLogCode);

IF iReadFB <> 0 THEN
	iReadFB.SetError();
END_IF
END_METHOD

METHOD PROTECTED ProcessResult : HRESULT
VAR_INPUT
	pResult	: POINTER TO SendDataRequestResult;
END_VAR
IF Valid THEN
	IF (CopyRemoteData(iObject, ePropID, pData, nData, pResult^.pData, pResult^.nData)) THEN
		IF iReadFB <> 0 THEN
			iReadFB.SetReady();
		END_IF
		ProcessResult:=S_OK;
	ELSE
		IF iReadFB <> 0 THEN
			iReadFB.SetError();
		END_IF
		ProcessResult:=E_FAIL;
	END_IF
END_IF
END_METHOD

METHOD GetRequestType : E_BACnetRM_RequestType
VAR_INPUT
END_VAR
GetRequestType:=E_BACnetRM_RequestType.eRead;
END_METHOD

END_FUNCTION_BLOCK

// POUs/Remote/Requests/[Internal]/FB_BACnetRM_ReqWpm
{attribute 'c++_compatible'}
{attribute 'enable_dynamic_creation'}
{attribute 'hide'}
FUNCTION_BLOCK FB_BACnetRM_ReqWpm EXTENDS FB_BACnetRM_ReqBasic
VAR_INPUT
	pEntries : POINTER TO ST_BACnetRM_WriteEntry;
	nEntries : UDINT;
	bFreeEntries : BOOL; 
END_VAR
VAR_OUTPUT
	bInit : BOOL;
END_VAR
VAR 
	{attribute 'hide'}
	req : SendDataRequest;
	{attribute 'hide'}
	pTmp : POINTER TO ST_BACnetRM_RpmListEntry;
END_VAR

IF NOT __ISVALIDREF(Client) THEN
	bError:=TRUE;
END_IF

SUPER^();

{attribute 'hide'}
METHOD Send : BOOL
IF Valid THEN
	IF stReq = 0 THEN
		Send:=FALSE;
		RETURN;
	END_IF
	
	UpdateRequest();
	Send:=SUPER^.Send();
END_IF
END_METHOD

METHOD INTERNAL UpdateRequest : BOOL
VAR_INPUT
END_VAR
VAR
	nSize : UDINT;
	i : UDINT;
	nTmpSize : UDINT;
	nTmpEntrySize : UDINT;
END_VAR
IF Valid THEN
	IF stReq <> 0 AND_THEN stReq^.pData <> 0 THEN
		pTmp:=stReq^.pData;
		__DELETE(pTmp);
	END_IF
	FOR i:=0 TO nEntries-1 DO
		IF pEntries[i].pEnable = 0 OR_ELSE pEntries[i].pEnable^ > 0 THEN
			nTmpSize := nTmpSize + SIZEOF(ST_BACnetRM_RpmListEntry) + F_BACnet_AlignedSize(F_BACnetRM_GetWriteEntrySize(pEntries[i]));
		END_IF
	END_FOR
	pTmp := __NEW(BYTE,nTmpSize);
	IF pTmp = 0 THEN
		UpdateRequest:=FALSE;
		RETURN;
	END_IF
	
	stReq := ADR(req);
	stReq^.pData := pTmp;
	FOR i:=0 TO nEntries-1 DO
		IF pEntries[i].pEnable = 0 OR_ELSE pEntries[i].pEnable^ > 0 THEN
			pTmp^.tObjectID := pEntries[i].iObject.ObjectID;
			pTmp^.ePropID := pEntries[i].ePropID;
			pTmp^.nArrayIndex := 0;
			pTmp^.nValidBits := 0; 
			IF pEntries[i].nPriority <> 16 THEN
				pTmp^.nValidBits.1 := 1;
				pTmp^.nPriority := pEntries[i].nPriority;
			ELSE
				pTmp^.nPriority := 0;
			END_IF
			nTmpEntrySize := F_BACnetRM_GetWriteEntrySize(pEntries[i]);
			pTmp^.nEntrySize := F_BACnet_AlignedSize(nTmpEntrySize) + SIZEOF(ST_BACnetRM_RpmListEntry) - 8;
			
			IF nTmpEntrySize <> 0 THEN
				MEMCPY(F_BACnet_EndOf(pTmp, SIZEOF(ST_BACnetRM_RpmListEntry)), pEntries[i].pData, pEntries[i].nData); 
			END_IF

			IF i <> nEntries -1 THEN
				pTmp[i].nEntrySize := pTmp[i].nEntrySize + 16#80000000;
			END_IF
			pTmp := F_BACnet_NextListElem(pTmp, pTmp^.nEntrySize);
		END_IF
	END_FOR
	
	stReq^.nData := nTmpSize;
	stReq^.service := E_BACnetConfirmedService.SrvWritePropertyMultiple;
	stReq^.deviceId := Client.ObjectInstance;
	
	bInit:=TRUE;
	
	UpdateRequest:=TRUE;
ELSE
	F_BA_LogMessage(ADSLOG_MSGTYPE_ERROR, 'WPM82', 'WPM Request not valid!');
END_IF
END_METHOD

METHOD PRIVATE Free
VAR_INPUT
END_VAR
IF bFreeEntries AND pEntries <> 0 THEN
	__DELETE(pEntries);
	pEntries:=0;
	bFreeEntries:=FALSE;
END_IF

IF stReq <> 0 AND_THEN stReq^.pData <> 0 THEN
	pTmp:=req.pData;
	__DELETE(pTmp);
	req.pData:=0;
	stReq:=0;
END_IF
END_METHOD

METHOD PROTECTED OnError
VAR_INPUT
	stResult		: POINTER TO SendDataRequestResult;
	sLogCode		: STRING			:= '';
END_VAR
VAR
	i : UDINT;
END_VAR
// Do not call super! Handle each entry's error:
// SUPER^.OnError(eResult, sLogCode);

FOR i:=0 TO nEntries-1 DO
	IF pEntries[i].iWriteFB <> 0 THEN
		pEntries[i].iWriteFB.SetError();
		IF (pEntries[i].iObject <> 0) THEN
			pEntries[i].iObject.OnReqError(THIS^, stResult, 'OE10');
		END_IF		
	END_IF
END_FOR
END_METHOD

METHOD PROTECTED ProcessResult : HRESULT
VAR_INPUT
	pResult	: POINTER TO SendDataRequestResult;
END_VAR
VAR
	pPropList : POINTER TO ST_BACnetRM_RpmListEntry;
END_VAR
VAR
	i : UDINT;
END_VAR
IF pResult^.service <> E_BACnetConfirmedService.SrvWritePropertyMultiple THEN
	SetError();
	RETURN;
END_IF

FOR i:=0 TO nEntries-1 DO
	IF pEntries[i].iWriteFB <> 0 THEN
		pEntries[i].iWriteFB.SetReady();	// TODO: handle error entry		
	END_IF
END_FOR
SetReady();
END_METHOD

METHOD GetRequestType : E_BACnetRM_RequestType
VAR_INPUT
END_VAR
GetRequestType := E_BACnetRM_RequestType.eWritePropertyMultiple;
END_METHOD

METHOD FB_exit : BOOL
VAR_INPUT
	bInCopyCode : BOOL; // if TRUE, the exit method is called for exiting an instance that is copied afterwards (online change).
END_VAR
Free();
END_METHOD

END_FUNCTION_BLOCK

// POUs/Remote/Requests/[Internal]/FB_BACnetRM_ReqWrite
{attribute 'c++_compatible'}
{attribute 'enable_dynamic_creation'}
{attribute 'hide'}
FUNCTION_BLOCK FB_BACnetRM_ReqWrite EXTENDS FB_BACnetRM_ReqBasic
VAR_INPUT CONSTANT
	ePropID : E_BACnetPropIdentifier;
	pData : PVOID;
	nData : UDINT;
	pEnable : POINTER TO BOOL;
	pNull : POINTER TO BOOL;
	fCOVIncrement : REAL;
	ePriority : E_BACnet_Priority := E_BACnet_Priority.Last;
	{attribute 'hide'}
	iWriteFB : I_BACnetRM_BasicReq;
END_VAR
VAR 
	{attribute 'hide'}
	req : SendDataRequest;
	{attribute 'hide'}
	lastWriteValue : ST_BACnetRM_LastWriteValue;
	{attribute 'hide'}
	bInstData : UDINT;
END_VAR
VAR_STAT
	{region 'Temporary'}
		{attribute 'hide'}
		_bEn : POINTER TO BOOL;
	{endregion}	
END_VAR

IF NOT __ISVALIDREF(Client) THEN
	bError:=TRUE;
END_IF

SUPER^();

{attribute 'hide'}
METHOD Send : BOOL
VAR
END_VAR
IF Valid THEN
	IF (pData <> 0) THEN
		IF stReq = 0 THEN
			req.service := E_BACnetConfirmedService.SrvWriteProperty;
			req.objectIdentifier := iObject.ObjectID;
			req.propertyIdentifier := ePropID;
			IF (F_BACnet_IsPriorityValid(ePriority)) THEN
				req.priority := TO_UDINT(ePriority);
			END_IF
			req.pData := pData;
			req.nData := nData;
			req.deviceId := Client.ObjectInstance;
			stReq := ADR(req);
		END_IF
		
		IF pNull <> 0 AND_THEN pNull^ THEN
			req.nData := 0;
		ELSE
			req.nData := nData;
		END_IF
		
		IF SUPER^.Send() THEN
			IF pNull <> 0 THEN
				lastWriteValue.stCmdValue.bNull := pNull^;
				IF nData <= 4 THEN
					MEMCPY(ADR(lastWriteValue.stCmdValue.fValue), pData, nData);
				ELSIF lastWriteValue.nOther <> 0 THEN
					MEMCPY(lastWriteValue.nOther, pData, nData);
				END_IF
			ELSE
				IF nData <= 4 THEN
					MEMCPY(ADR(lastWriteValue.n32Value), pData, nData);
				ELSIF lastWriteValue.nOther <> 0 THEN
					MEMCPY(lastWriteValue.nOther, pData, nData);
				END_IF
			END_IF
			Send:=TRUE;
		END_IF
	END_IF
END_IF
END_METHOD

METHOD PROTECTED OnError
VAR_INPUT
	stResult		: POINTER TO SendDataRequestResult;
	sLogCode		: STRING			:= '';
END_VAR
SUPER^.OnError(stResult, sLogCode);

IF iWriteFB <> 0 THEN
	iWriteFB.SetError();
END_IF
END_METHOD

METHOD PROTECTED ProcessResult : HRESULT
VAR_INPUT
	pResult	: POINTER TO SendDataRequestResult;
END_VAR
bReady:=TRUE;

IF iWriteFB <> 0 THEN
	iWriteFB.SetReady();
END_IF

ProcessResult:=S_OK;
END_METHOD

METHOD GetRequestType : E_BACnetRM_RequestType
VAR_INPUT
END_VAR
GetRequestType := E_BACnetRM_RequestType.eWrite;
END_METHOD

METHOD IsReady : BOOL
VAR_INPUT
END_VAR
VAR
	_fValue : REAL;
END_VAR
IF SUPER^.IsReady() THEN
	IF pEnable = 0 OR_ELSE pEnable^ THEN		
		IF fCOVIncrement <> 0.0 THEN
			MEMCPY(ADR(_fValue), pData, SIZEOF(_fValue));
			IF ABS(lastWriteValue.stCmdValue.fValue - _fValue) > fCOVIncrement THEN
				IF pNull = 0 OR_ELSE NOT pNull^ THEN
					IsReady:=TRUE;
					RETURN;
				END_IF
			END_IF
		ELSE
			IF MEMCMP(ADR(lastWriteValue.n32Value), pData, nData) <> 0 THEN 
				IF pNull = 0 OR_ELSE NOT pNull^ THEN
					IsReady:=TRUE;
					RETURN;
				END_IF
			END_IF
		END_IF
		IF pNull <> 0 AND_THEN pNull^ <> lastWriteValue.stCmdValue.bNull THEN
			IsReady:=TRUE;
			RETURN;
		END_IF
	END_IF
END_IF
END_METHOD

END_FUNCTION_BLOCK

// POUs/Remote/Properties/FB_BACnetRM_ReadProperty
FUNCTION_BLOCK FB_BACnetRM_ReadProperty EXTENDS FB_BACnetRM_BaseProperty
VAR_INPUT CONSTANT
	{attribute 'initialize_on_call'}
	{attribute 'no_copy'}
	Client : REFERENCE TO FB_BACnet_Client;
	bReqRPM : BOOL;
END_VAR

SUPER^();

METHOD PROTECTED OnExecuteChange : BOOL
OnExecuteChange := Client.AddFifoReadReq(THIS);
END_METHOD

METHOD PROTECTED Free : BOOL
IF pRequest.pPtr <> 0 THEN
	IF bReqRPM AND pRequest.fbRpm <> 0 THEN
		__DELETE(pRequest.fbRpm);
		pRequest.fbRpm:=0;
	ELSIF pRequest.fbRead <> 0 THEN
		__DELETE(pRequest.fbRead);
		pRequest.fbRead:=0;
	END_IF
	pRequest.pPtr:=0;
END_IF
END_METHOD

PROPERTY Valid : BOOL
GET
Valid := __ISVALIDREF(Client);
END_GET
END_PROPERTY

METHOD FB_exit : BOOL
VAR_INPUT
	bInCopyCode : BOOL; // if TRUE, the exit method is called for exiting an instance that is copied afterwards (online change).
END_VAR
Free();
END_METHOD

END_FUNCTION_BLOCK

// POUs/Remote/Properties/[Base]/FB_BACnetRM_BaseProperty
FUNCTION_BLOCK FB_BACnetRM_BaseProperty IMPLEMENTS I_BACnetRM_BasicReq
VAR_INPUT CONSTANT
	pData : PVOID;
	nData : UDINT;
	iObject : I_BACnetRM_BaseObject;
	nIndex : UDINT := 16#FFFFFFFF;
	ePropID : E_BACnetPropIdentifier;
	bExecute : BOOL;
	{attribute 'hide'}
	pRequest : ST_BACnetRM_ReqPtr;
END_VAR
VAR_OUTPUT
	bReady : BOOL;
	bBusy : BOOL;
	bError : BOOL;
END_VAR
VAR
	{attribute 'hide'}
	bExecuteOld : BOOL;
END_VAR

IF bExecuteOld <> bExecute THEN
	bExecuteOld := bExecute;

	IF NOT Valid THEN
		SetError();
	END_IF
	
	IF bExecute THEN
		IF bBusy THEN
			RETURN;
		END_IF
		Free();
		IF NOT OnExecuteChange() THEN
			SetError();
		ELSE
			SetBusy();
		END_IF
	ELSE
		bReady:=FALSE;
	END_IF
END_IF

{attribute 'hide'}
METHOD SetBusy
bBusy := TRUE;
bError := FALSE;
bReady := FALSE;
END_METHOD

{attribute 'hide'}
METHOD SetError
bBusy := FALSE;
bError := TRUE;
bReady := FALSE;
END_METHOD

{attribute 'hide'}
METHOD SetReady
bBusy := FALSE;
bError := FALSE;
bReady := TRUE;
END_METHOD

METHOD PROTECTED OnExecuteChange : BOOL
OnExecuteChange := FALSE;
END_METHOD

METHOD PROTECTED Free : BOOL
Free := FALSE;
END_METHOD

PROPERTY Busy : BOOL
GET
Busy:=bBusy;
END_GET
SET
bBusy:=Busy;
END_SET
END_PROPERTY

PROPERTY Error : BOOL
GET
Error:=bError;
END_GET
SET
bError:=Error;
END_SET
END_PROPERTY

PROPERTY Ready : BOOL
GET
Ready:=bReady;
END_GET
SET
bReady:=Ready;
END_SET
END_PROPERTY

PROPERTY Request : ST_BACnetRM_ReqPtr;
GET
Request:=pRequest;
END_GET
SET
pRequest:=Request;
END_SET
END_PROPERTY

PROPERTY Valid : BOOL
GET
Valid := FALSE;
END_GET
END_PROPERTY

END_FUNCTION_BLOCK

// POUs/Remote/Properties/FB_BACnetRM_WriteProperty
FUNCTION_BLOCK FB_BACnetRM_WriteProperty EXTENDS FB_BACnetRM_BaseProperty
VAR_INPUT CONSTANT
	{attribute 'initialize_on_call'}
	{attribute 'no_copy'}
	Client : REFERENCE TO FB_BACnet_Client;
	
	bRequestWPM : BOOL;
END_VAR

SUPER^();

METHOD PROTECTED OnExecuteChange : BOOL
OnExecuteChange := Client.AddFifoWriteReq(THIS);
END_METHOD

METHOD PROTECTED Free : BOOL
IF pRequest.pPtr <> 0 THEN
	IF bRequestWPM  AND pRequest.fbWpm <> 0 THEN
		__DELETE(pRequest.fbWpm);
		pRequest.fbWpm:=0;
	ELSIF pRequest.fbWrite <> 0 THEN
		__DELETE(pRequest.fbWrite);
		pRequest.fbWrite:=0;
	END_IF
	pRequest.pPtr:=0;
END_IF
END_METHOD

PROPERTY Valid : BOOL
GET
Valid := __ISVALIDREF(Client);
END_GET
END_PROPERTY

METHOD FB_exit : BOOL
VAR_INPUT
	bInCopyCode : BOOL; // if TRUE, the exit method is called for exiting an instance that is copied afterwards (online change).
END_VAR
Free();
END_METHOD

END_FUNCTION_BLOCK

// POUs/Remote/Requests/[Internal]/FB_BACnetRM_ReqCov
{attribute 'c++_compatible'}
{attribute 'enable_dynamic_creation'}
{attribute 'hide'}
{attribute 'hide'}
FUNCTION_BLOCK FB_BACnetRM_ReqCov EXTENDS FB_BACnetRM_ReqBasic
VAR_INPUT CONSTANT
	bConfirmed : BOOL;
	bUnsubscribed : BOOL;
	tLifetime : TIME := T#300S;
	fCOVIncrement : REAL := 0;
END_VAR
VAR_INPUT
	ePropID : E_BACnetPropIdentifier;
	pData : PVOID;
	nData : UDINT;
END_VAR
VAR_OUTPUT
	bSubsReady : BOOL;
END_VAR
VAR 
	req : SubscribeCovPropertyRequest;
	bSendSubs : BOOL := TRUE;
	pMaster : POINTER TO FB_BACnetRM_ReqCov;
	pCovSlaves : POINTER TO POINTER TO FB_BACnetRM_ReqCov;
	nCovSlaves : UDINT;
	nCovSlavesMax : UDINT;
END_VAR

IF NOT __ISVALIDREF(Client) THEN
	bError:=TRUE;
END_IF

SUPER^();

METHOD INTERNAL AddCovSlave : BOOL
VAR_INPUT
	pSlave : POINTER TO FB_BACnetRM_ReqCov;
END_VAR
VAR
	nTmp : UDINT;
	nTmpSize : UDINT;
	pTmp : POINTER TO POINTER TO FB_BACnetRM_ReqCov;
END_VAR
IF nCovSlaves+1 >= nCovSlavesMax THEN
	nTmp := nCovSlavesMax+10;
	nTmpSize := nTmp*SIZEOF(POINTER TO FB_BACnetRM_ReqCov);
	pTmp := __NEW(BYTE,nTmpSize);
	IF pTmp = 0 THEN
		RETURN;
	END_IF
	IF pCovSlaves <> 0 THEN
		MEMCPY(pTmp, pCovSlaves, nCovSlavesMax*SIZEOF(POINTER TO FB_BACnetRM_ReqCov));
		__DELETE(pCovSlaves);
	END_IF
	pCovSlaves:=pTmp;
	nCovSlavesMax:=nTmp;
END_IF

pCovSlaves[nCovSlaves]:=pSlave;
nCovSlaves:=nCovSlaves+1;
END_METHOD

{attribute 'hide'}
METHOD Send : BOOL
VAR
	iClientTmp : ITcIoBACnetPlcClient;
END_VAR
IF Valid THEN
	IF NOT bSendSubs THEN
		RETURN;
	END_IF
	
	IF stReq = 0 THEN
		IF bUnsubscribed THEN
			req.issueConfirmedNotifications := FALSE;
			req.lifetime := 0;
			req.subscriberProcessIdentifier := 0;
		ELSE
			req.issueConfirmedNotifications := bConfirmed;
			req.lifetime := TIME_TO_DWORD(tLifetime) / 500;
			req.subscriberProcessIdentifier := 1;
		END_IF
		req.monitoredObjectIdentifier := iObject.ObjectID;
		req.covIncrement := fCOVIncrement;
		req.monitoredPropertyIdentifier.propertyIdentifier := ePropID;
		req.monitoredPropertyIdentifier.validFields := 1;	
	
		req.validFields := 2#0011111;
		IF req.covIncrement <> 0 THEN
			req.validFields := req.validFields +  2#100000;
		END_IF
	END_IF
	
	iClientTmp := Client.iClient;
	IF S_OK = iClientTmp.SendCOVSubscription(ADR(req), THIS^) THEN
		Send:=TRUE;
		StartTimer();
	END_IF
END_IF
END_METHOD

METHOD PROTECTED ProcessResult : HRESULT
VAR_INPUT
	pResult	: POINTER TO SendDataRequestResult;
END_VAR
VAR
	pPropList : POINTER TO ST_BACnetRM_PropertyValueList;
	i : UDINT;
END_VAR
IF Valid THEN
	IF pResult^.service = E_BACnetConfirmedService.SrvSubscribeCOV OR pResult^.service = E_BACnetConfirmedService.SrvSubscribeCOVProperty THEN
		bSubsReady:=TRUE;
		RETURN;
	END_IF
	
	ProcessResult:=E_FAIL;
	
	IF pResult^.objectIdentifier = iObject.ObjectID THEN
		pPropList := pResult^.pData;
		WHILE pPropList <> 0 DO
			IF pPropList^.ePropID = ePropID THEN
				CopyRemoteData(iObject, ePropID, pData, nData, F_BACnet_EndOf(pPropList, SIZEOF(ST_BACnetRM_PropertyValueList)), pPropList^.nValueSize -  SIZEOF(DWORD));
				ProcessResult:=S_OK;
			END_IF
			pPropList := F_BACnet_NextListElem(pPropList, pPropList^.nEntrySize);
		END_WHILE
	END_IF
	
	IF pCovSlaves <> 0 AND nCovSlaves > 0 THEN
		FOR i:=0 TO nCovSlaves-1 DO
			pCovSlaves[i]^.ProcessResult(pResult);
		END_FOR
	END_IF
ELSE
	// (BETA) ... Output Error
END_IF
END_METHOD

METHOD PROTECTED StartTimer : BOOL
VAR_INPUT
END_VAR
timer(IN:=FALSE, PT:=tLifetime);
timer(IN:=TRUE, PT:=tLifetime);
END_METHOD

METHOD GetRequestType : E_BACnetRM_RequestType
VAR_INPUT
END_VAR
GetRequestType := E_BACnetRM_RequestType.eCov;
END_METHOD

METHOD IsReady : BOOL
VAR_INPUT
END_VAR
IF NOT bSendSubs THEN
	IsReady:=TRUE;
	RETURN;
END_IF

IsReady:=SUPER^.IsReady();
END_METHOD

METHOD FB_Exit : BOOL
VAR_INPUT
	 bInCopyCode : BOOL; // if TRUE, the exit method is called for exiting an instance that is copied afterwards (online change).
END_VAR
VAR
	i : UDINT;
END_VAR
IF pCovSlaves <> 0 THEN
	__DELETE(pCovSlaves);
	pCovSlaves:=0;
END_IF
pMaster:=0;
END_METHOD

PROPERTY Master : POINTER TO FB_BACnetRM_ReqCov
GET
Master:=pMaster;
END_GET
SET
pMaster:=Master;
END_SET
END_PROPERTY

PROPERTY SendSubscription : BOOL
GET
SendSubscription:=bSendSubs;
END_GET
SET
bSendSubs:=SendSubscription;
END_SET
END_PROPERTY

END_FUNCTION_BLOCK

// POUs/Remote/Objects/Basic/FB_BACnetRM_AV
{attribute 'enable_dynamic_creation'}
FUNCTION_BLOCK FB_BACnetRM_AV EXTENDS FB_BACnetRM_EventObject
VAR_INPUT
	bEnWrite 		: BOOL;
	fVal 			: REAL;
	bNullVal 		: BOOL;	
END_VAR
VAR_INPUT CONSTANT PERSISTENT
	{region 'Fixed Parameters'}
		{attribute 'parameterCategory':='Config'}
		fReadIncrement : REAL; 
		{attribute 'parameterCategory':='Config'}
		fWriteIncrement : REAL; 
			 
		{attribute 'parameterCategory':='Value'}
		ePriority 	  : E_BACnet_Priority := BACnet_Param.eRemotePrio_Default;
	{endregion}
END_VAR
VAR_OUTPUT
	fPresVal 	: REAL;
END_VAR

SUPER^();

METHOD PROTECTED OnObjectStateChanged
SUPER^.OnObjectStateChanged();

SyncPropertyReal(E_BACnetPropIdentifier.PropPresentValue, SIZEOF(fPresVal), ADR(fPresVal), E_BA_SyncModeRM.eRead, fReadIncrement);

SyncPropertyPrioReal(E_BACnetPropIdentifier.PropPresentValue, SIZEOF(fVal), ADR(fVal), ADR(bEnWrite), ADR(bNullVal), ePriority, E_BA_SyncModeRM.eWrite, fWriteIncrement);
END_METHOD

